    // After move finishes, check abort status and flags
    5:
        IF fbMotionStage.ExMotionStatus.bIdling THEN
            AssertTrue(
                Condition := fbMotionStage.ExMotionStatus.bAborted,
                Message   := 'Move must be aborted #8'
            );
            AssertFalse(
                Condition := fbMotionStage.stMotionStatus.bBusy,
                Message   := 'Move request must be canceled #9'
            );
            AssertFalse(
                Condition := fbMotionStage.stExMotionStatus.bExecute,
                Message   := 'Move request must cleared #10'
            );
            nTestStep := 6;
        END_IF	
END_CASE

// Cyclically call timer FBs
fbTestTimer();
fbAbsoluteMoveHaltTimer();

// End test or handle timeout
IF nTestStep = 6 THEN
    TEST_FINISHED();
ELSIF fbTestTimer.Q THEN
    AssertTrue(
        Condition := FALSE,
        Message := CONCAT('Timed out at step: ', TO_STRING(nTestStep))
    );
    TEST_FINISHED();
END_IF
END_METHOD

METHOD PRIVATE GivenMoveCmdAndMoveOkIfResetThenAbortMove_Test1
VAR_INST
   fbMotionStage : FB_MotionStageNC(	sName := 'TEST1',
                                        AxisRef := fbAxisRef[1],
                                        iPersistentDataStorage := fbPersistentDataStorage[1]
                                    ):=(SaveAxisParams := FALSE);
									
    fbTestTimer: TON := (IN:=TRUE, PT:=T#3S);
    fbAbsoluteMoveResetTimer: TON := (PT:=T#500MS);
    nTestStep : INT;
END_VAR
TEST(__POUNAME());

// motion stage block
fbMotionStage();

// Main test state machine
CASE nTestStep OF
    // === Interlock Fault Test ===
    0:
        IF fbMotionStage.ExMotionStatus.bInterlocksError THEN
            AssertTrue(
                Condition := fbMotionStage.stMotionStatus.bError,
                Message := 'Interlock error must be raised #1'
            );
            AssertEquals_UDINT(
                Expected := 11,
                Actual := fbMotionStage.stMotionStatus.nErrorId,
                Message := 'Interlock error code is 11 #2'
            );
        END_IF
        nTestStep := nTestStep + 1;
    
    // === Reset and Enable Features ===
    1:
        fbMotionStage.Reset();
        fbMotionStage.EnableLimits(
			BackwardEnable:=TRUE, 
			ForwardEnable:=TRUE,
			HomeEnable:=FALSE
		);
        fbMotionStage.EnableInterlocks();
        // Note: Trying to write to a property with 'GET' only should fail! See notes below.
        // fbMotionStage.MotionStatus.bExecute := TRUE; // Should be forbidden if it's a read-only property

        nTestStep := nTestStep + 1;    

    // === Abort Done/Status Check ===
    2:
        IF fbMotionStage.ExMotionStatus.bAbortDone THEN
            AssertFalse(
                Condition := fbMotionStage.stMotionStatus.bError,
                Message := 'Error must be cleared #3'
            );
            AssertEquals_UDINT(
                Expected := 0,
                Actual := fbMotionStage.stMotionStatus.nErrorId,
                Message := 'error ID must be 0 #4'
            );
            nTestStep := nTestStep + 1;    
        END_IF

    // === Absolute Move Request ===
    3:
        fbMotionStage.AbsoluteMove(
            Position := 10000.0,
            Velocity := 50.0,
            Acceleration := 500.0,
            Deceleration := 500.0
        );
        fbAbsoluteMoveResetTimer.IN := TRUE;
        nTestStep := nTestStep + 1;

    // === Move Reset after Timer ===
    4:
        IF fbAbsoluteMoveResetTimer.Q THEN
            fbMotionStage.Reset();
            fbAbsoluteMoveResetTimer.IN := FALSE;
            nTestStep := nTestStep + 1;
        END_IF

    // === Move Done/Abort Confirmation ===
    5:
        IF fbMotionStage.stExMotionStatus.bAbortDone THEN
            nTestStep := nTestStep + 1;
        END_IF
	6:
		IF fbMotionStage.stExMotionStatus.bAborted THEN
            AssertFalse(
                Condition := fbMotionStage.stMotionStatus.bBusy,
                Message := 'Move request must be canceled #6'
            );
            AssertFalse(
                Condition := fbMotionStage.stExMotionStatus.bExecute,
                Message := 'Move request must be cleared #7'
            );
            nTestStep := nTestStep + 1;
		END_IF
END_CASE

// Update timers
fbTestTimer();
fbAbsoluteMoveResetTimer();

// Test Completion Handlers
IF nTestStep = 7 THEN
    TEST_FINISHED();
ELSIF fbTestTimer.Q THEN
    AssertTrue(
        Condition := FALSE,
        Message := CONCAT('Timed out at step: ', TO_STRING(nTestStep))
    );
    TEST_FINISHED();
END_IF
END_METHOD

METHOD PRIVATE GivenMoveCmdAndMoveOkMoveToTarget1ThenTarget2_Test3
VAR_INST
   fbMotionStage : FB_MotionStageNC(	sName := 'Test3',
                                        AxisRef := fbAxisRef[3],
                                        iPersistentDataStorage := fbPersistentDataStorage[3]
                                    ):=(SaveAxisParams := FALSE);
									
    fbTestTimer: TON := (IN:=TRUE, PT:=T#10S);
    nTestStep : INT;
END_VAR
TEST(__POUNAME());

CASE nTestStep OF
    0: // Enable safety interlocks and hardware limits
        fbMotionStage.EnableLimits(
			BackwardEnable:=TRUE, 
			ForwardEnable:=TRUE,
			HomeEnable:=FALSE
		);
        fbMotionStage.EnableInterlocks();
        nTestStep := 1;

    1: // Issue initial absolute move to position 100.0 with no backlash
        fbMotionStage.AbsoluteMove(
            Position := 100.0,
            Velocity := 50.0,
            Acceleration := 500.0,
            Deceleration := 500.0
        );
        nTestStep := 2;

    2: // Wait for move done
        IF fbMotionStage.stMotionStatus.bDone THEN
            AssertTrue(
                Condition := ABS(fbMotionStage.MotionCmd.fPosition - fbAxisRef[3].NcToPlc.ActPos) < 0.001,
                Message := 'Target position not reached #1'
            );
            nTestStep := 3;
        END_IF

    3: // When idling, perform another absolute move
        IF fbMotionStage.ExMotionStatus.bIdling THEN
            fbMotionStage.AbsoluteMove(
                Position := 320.0,
                Velocity := 50.0,
                Acceleration := 500.0,
                Deceleration := 500.0
            );
            nTestStep := 4;
        END_IF

    4: // Wait for second move done
        IF fbMotionStage.stMotionStatus.bDone THEN
            AssertTrue(
                Condition := ABS(fbMotionStage.MotionCmd.fPosition - fbAxisRef[3].NcToPlc.ActPos) < 0.001,
                Message := 'Target position not reached #2'
            );
            nTestStep := 5;
          END_IF

END_CASE

fbTestTimer();
fbMotionStage();

IF nTestStep = 5 THEN
    TEST_FINISHED();
ELSIF fbTestTimer.Q THEN
    AssertTrue(
        Condition := FALSE,
        Message := CONCAT('Timed out at step: ', TO_STRING(nTestStep))
    );
    TEST_FINISHED();
END_IF
END_METHOD

METHOD PRIVATE GivenMoveCmdAndValidInterlocksThenMoveToTarget_Test4
VAR_INST
   fbMotionStage : FB_MotionStageNC(	sName := 'Test4',
                                        AxisRef := fbAxisRef[4],
                                        iPersistentDataStorage := fbPersistentDataStorage[4]
                                    ):=(SaveAxisParams := FALSE);
									
    fbTestTimer: TON := (IN:=TRUE, PT:=T#3S);
    nTestStep : INT;
END_VAR
TEST(__POUNAME());

CASE nTestStep OF
    0: // Enable safety interlocks and hardware limits
        fbMotionStage.EnableLimits(
			BackwardEnable:=TRUE, 
			ForwardEnable:=TRUE,
			HomeEnable:=FALSE
		);
        fbMotionStage.EnableInterlocks();
        nTestStep := 1;

    1: // Issue initial absolute move to position 100.0 with no backlash
        fbMotionStage.AbsoluteMove(
            Position := 100.0,
            Velocity := 50.0,
            Acceleration := 500.0,
            Deceleration := 500.0
        );
        nTestStep := 2;

    2: // Wait for move done
        IF fbMotionStage.stMotionStatus.bDone THEN
            AssertTrue(
                Condition := ABS(fbMotionStage.MotionCmd.fPosition - fbAxisRef[4].NcToPlc.ActPos) < 0.001,
                Message := 'Target position not reached #1'
            );
            nTestStep := 3;
        END_IF
END_CASE

fbTestTimer();
fbMotionStage();

IF nTestStep = 3 THEN
    TEST_FINISHED();
ELSIF fbTestTimer.Q THEN
    AssertTrue(
        Condition := FALSE,
        Message := CONCAT('Timed out at step: ', TO_STRING(nTestStep))
    );
    TEST_FINISHED();
END_IF
END_METHOD

METHOD PRIVATE GivenMoveCmdValidInterlockAndWrongMotionParamsThenGotoErrorStateIfResetThenGotoInitState_Test5
VAR_INST
   fbMotionStage : FB_MotionStageNC(	sName := 'Test5',
                                        AxisRef := fbAxisRef[5],
                                        iPersistentDataStorage := fbPersistentDataStorage[5]
                                    ):=(SaveAxisParams := FALSE);
									
    fbTestTimer: TON := (IN:=TRUE, PT:=T#3S);
    fbAbsoluteMoveTimer: TON := (PT:=T#50MS);
    nTestStep : INT;
END_VAR
TEST(__POUNAME());

CASE nTestStep OF
    0:
        fbMotionStage.EnableLimits(
			BackwardEnable:=TRUE, 
			ForwardEnable:=TRUE,
			HomeEnable:=FALSE
		);
        fbMotionStage.EnableInterlocks();
        nTestStep := 1;
	1:// Issue initial absolute move to position 100.0 with no backlash
        fbMotionStage.AbsoluteMove(
            Position := 100.0,
            Velocity := 0.0,
            Acceleration := 500.0,
            Deceleration := 500.0
        );
		nTestStep := 2;
	2:
		IF (fbMotionStage.stExMotionStatus.eDriveState=E_MoveState.ERROR) THEN
			nTestStep := 3;
		END_IF
END_CASE
fbMotionStage();
fbTestTimer();
fbAbsoluteMoveTimer();


IF nTestStep = 3 THEN

TEST_FINISHED();
ELSIF fbTestTimer.Q THEN
    AssertTrue(
        Condition := FALSE,
        Message := CONCAT('Timed out at step: ', TO_STRING(nTestStep))
    );
    TEST_FINISHED();
END_IF
END_METHOD

METHOD PRIVATE OverallStageFeaturesAndOperationalTests_Test17
VAR_INST
   fbMotionStage : FB_MotionStageNC(	sName := 'Test17',
                                        AxisRef := fbAxisRef[17],
                                        iPersistentDataStorage := fbPersistentDataStorage[17]
                                    ) := (SaveAxisParams := FALSE);
									
    fbTestTimer: TON := (IN:=TRUE, PT:=T#180S);
    fbResetTimer: TON := (IN:=FALSE, PT:=T#500MS);;
	fbInMotionTimer : TON := (IN:=FALSE, PT:=T#800MS);;
    fbCamSwitchPulserSearch : TON := (IN:=FALSE, PT:=T#1000MS);
    fbCamSwitchPulserSync: TON := (IN:=FALSE, PT:=T#2000MS);
    nTestStep : INT;
END_VAR
TEST(__POUNAME());

CASE nTestStep OF

/// ------------ INITIAL SETUP ---------------
0:
    fbMotionStage.EnableLimits(
        BackwardEnable := TRUE, ForwardEnable := TRUE, HomeEnable := FALSE);
    fbMotionStage.EnableInterlocks();
    nTestStep := 1;

/// ------- 3 FAST ABSOLUTE MOVES ------------
/// (All moves <= 50 units, velocities set for sub-second moves)
1:
    fbMotionStage.AbsoluteMove(Position := 10.0, Velocity := 50.0, Acceleration := 200.0, Deceleration := 200.0);
    nTestStep := 2;
2:
    IF fbMotionStage.stMotionStatus.bDone THEN
        AssertTrue(ABS(10.0 - fbAxisRef[17].NcToPlc.ActPos) < 0.01, 'Move#1');
        nTestStep := 3;
    END_IF
3:
    fbMotionStage.AbsoluteMove(Position := -8.0, Velocity := 50.0, Acceleration := 200.0, Deceleration := 200.0);
    nTestStep := 4;
4:
    IF fbMotionStage.stMotionStatus.bDone THEN
        AssertTrue(ABS(-8.0 - fbAxisRef[17].NcToPlc.ActPos) < 0.01, 'Move#2');
        nTestStep := 5;
    END_IF
5:
    fbMotionStage.AbsoluteMove(Position := 15.0, Velocity := 50.0, Acceleration := 150.0, Deceleration := 150.0);
    nTestStep := 6;
6:
    IF fbMotionStage.stMotionStatus.bDone THEN
        AssertTrue(ABS(15.0 - fbAxisRef[17].NcToPlc.ActPos) < 0.01, 'Move#3');
        nTestStep := 7;
    END_IF

/// -------- HALT and RESET POS/NEG ------------

7:
    fbMotionStage.AbsoluteMove(Position := 18.0, Velocity := 70.0, Acceleration := 200.0, Deceleration := 200.0);
    fbInMotionTimer.PT := T#120MS;
    fbInMotionTimer.IN := TRUE;
    nTestStep := 8;
8:
    IF fbMotionStage.stMotionStatus.bBusy AND fbInMotionTimer.Q THEN
        fbMotionStage.Halt();
        fbInMotionTimer.IN := FALSE;
        nTestStep := 9;
    END_IF
9:
    IF fbMotionStage.stExMotionStatus.bAborted THEN
        AssertFalse(fbMotionStage.stMotionStatus.bBusy, 'Halt busy/fwd');
        nTestStep := 10;
    END_IF

10:
    fbMotionStage.AbsoluteMove(Position := -12.0, Velocity := 70.0, Acceleration := 200.0, Deceleration := 200.0);
    fbInMotionTimer.PT := T#120MS;
    fbInMotionTimer.IN := TRUE;
    nTestStep := 11;
11:
    IF fbMotionStage.stMotionStatus.bBusy AND fbInMotionTimer.Q THEN
        fbMotionStage.Halt();
        fbInMotionTimer.IN := FALSE;
        nTestStep := 12;
    END_IF
12:
    IF fbMotionStage.stExMotionStatus.bAborted THEN
        AssertFalse(fbMotionStage.stMotionStatus.bBusy, 'Halt busy/bwd');
        nTestStep := 13;
    END_IF

13:
    fbMotionStage.AbsoluteMove(Position := 21.0, Velocity := 70.0, Acceleration := 200.0, Deceleration := 200.0);
    fbInMotionTimer.PT := T#120MS;
    fbInMotionTimer.IN := TRUE;
    nTestStep := 14;
14:
    IF fbMotionStage.stMotionStatus.bBusy AND fbInMotionTimer.Q THEN
        fbMotionStage.Reset();
        fbInMotionTimer.IN := FALSE;
        nTestStep := 15;
    END_IF
15:
    IF fbMotionStage.stExMotionStatus.bAborted THEN
        AssertFalse(fbMotionStage.stMotionStatus.bBusy, 'Reset busy/fwd');
        nTestStep := 16;
    END_IF

16:
    fbMotionStage.AbsoluteMove(Position := -22.0, Velocity := 70.0, Acceleration := 200.0, Deceleration := 200.0);
    fbInMotionTimer.PT := T#120MS;
    fbInMotionTimer.IN := TRUE;
    nTestStep := 17;
17:
    IF fbMotionStage.stMotionStatus.bBusy AND fbInMotionTimer.Q THEN
        fbMotionStage.Reset();
        fbInMotionTimer.IN := FALSE;
        nTestStep := 18;
    END_IF
18:
    IF fbMotionStage.stExMotionStatus.bAborted THEN
        AssertFalse(fbMotionStage.stMotionStatus.bBusy, 'Reset busy/bwd');
        nTestStep := 19;
    END_IF

/// -------- LIMIT HIT TEST (FORWARD THEN BACKWARD) ----------
19:
    fbMotionStage.AbsoluteMove(Position := 25.0, Velocity := 50.0, Acceleration := 120.0, Deceleration := 120.0);
    fbInMotionTimer.PT := T#120MS; fbInMotionTimer.IN := TRUE; nTestStep := 20;
20:
    IF fbMotionStage.stMotionStatus.bBusy AND fbInMotionTimer.Q THEN
        fbMotionStage.EnableLimits(BackwardEnable := TRUE, ForwardEnable := FALSE, HomeEnable := FALSE);
        fbInMotionTimer.IN := FALSE; nTestStep := 21;
    END_IF
21:
    IF fbMotionStage.stMotionStatus.bWarning AND fbMotionStage.stExMotionStatus.bAborted THEN
        fbMotionStage.EnableLimits(BackwardEnable := TRUE, ForwardEnable := TRUE, HomeEnable := FALSE);
        nTestStep := 22;
    END_IF
22: nTestStep := 23;

23:
    fbMotionStage.AbsoluteMove(Position := -25.0, Velocity := 50.0, Acceleration := 120.0, Deceleration := 120.0);
    fbInMotionTimer.PT := T#120MS; fbInMotionTimer.IN := TRUE; nTestStep := 24;
24:
    IF fbMotionStage.stMotionStatus.bBusy AND fbInMotionTimer.Q THEN
        fbMotionStage.EnableLimits(BackwardEnable := FALSE, ForwardEnable := TRUE, HomeEnable := FALSE);
        fbInMotionTimer.IN := FALSE; nTestStep := 25;
    END_IF
25:
    IF fbMotionStage.stMotionStatus.bWarning AND fbMotionStage.stExMotionStatus.bAborted THEN
        fbMotionStage.EnableLimits(BackwardEnable := TRUE, ForwardEnable := TRUE, HomeEnable := FALSE);
        nTestStep := 26;
    END_IF
26: nTestStep := 27;

/// ------------- Home+Move Alternation: All major home modes ------------
/// (Home, then absolute move. All positions ~10-30 units, velocities >= 50.)
27:
    fbMotionStage.Home(HomePosition := 10.0, HomeMode := E_EpicsHomeCmd.LOW_LIMIT);
    fbCamSwitchPulserSearch.IN := TRUE; nTestStep := 28;
28:
    IF fbCamSwitchPulserSearch.Q THEN
        fbMotionStage.EnableLimits(BackwardEnable := FALSE, ForwardEnable := TRUE, HomeEnable := FALSE);
        fbCamSwitchPulserSearch.IN := FALSE; fbCamSwitchPulserSync.IN := TRUE;
        nTestStep := 29;
    END_IF
29:
    IF fbCamSwitchPulserSync.Q THEN
        fbMotionStage.EnableLimits(BackwardEnable := TRUE, ForwardEnable := TRUE, HomeEnable := FALSE);
        fbCamSwitchPulserSync.IN := FALSE; nTestStep := 30;
    END_IF
30:
    IF fbMotionStage.stMotionStatus.bDone THEN
        AssertTrue(fbAxisRef[17].Status.Homed, 'Home#1 (LOW_LIMIT): Axis not calibrated'); 
		AssertEquals_LREAL(Delta := 0.001, Expected := 10.0, Actual := fbAxisRef[17].NcToPlc.ActPos, Message :='Home#1: Not at expected home');
        nTestStep := 31;
    END_IF
31: 
	fbMotionStage.AbsoluteMove(Position := 20.0, Velocity := 50.0, Acceleration := 200.0, Deceleration := 200.0);
	nTestStep := 32;
32: 
	IF fbMotionStage.stMotionStatus.bDone THEN
		AssertTrue(ABS(20.0 - fbAxisRef[17].NcToPlc.ActPos) < 0.01, 'Move#4: Target position not reached after home');
		nTestStep := 33;
	END_IF

33: 
	fbMotionStage.Home(HomePosition := 25.0, HomeMode := E_EpicsHomeCmd.HIGH_LIMIT);
	fbCamSwitchPulserSearch.IN := TRUE; 
	nTestStep := 34;
34: 
	IF fbCamSwitchPulserSearch.Q THEN 
		fbMotionStage.EnableLimits(BackwardEnable := TRUE, ForwardEnable := FALSE, HomeEnable := FALSE);
		fbCamSwitchPulserSearch.IN := FALSE;
		fbCamSwitchPulserSync.IN := TRUE;
		nTestStep := 35;
	END_IF
35: 
	IF fbCamSwitchPulserSync.Q THEN
		fbMotionStage.EnableLimits(BackwardEnable := TRUE, ForwardEnable := TRUE, HomeEnable := FALSE);
		fbCamSwitchPulserSync.IN := FALSE;
		nTestStep := 36;
	END_IF
36: 
	IF fbMotionStage.stMotionStatus.bDone THEN 
		AssertTrue(fbAxisRef[17].Status.Homed, 'Home#2 (HIGH_LIMIT): Axis not calibrated');
		AssertEquals_LREAL(Delta := 0.001, Expected := 25.0, Actual := fbAxisRef[17].NcToPlc.ActPos, Message := 'Home#2: Not at expected home'); 
		nTestStep := 37; 
	END_IF
37: 
	fbMotionStage.AbsoluteMove(Position := -20.0, Velocity := 50.0, Acceleration := 200.0, Deceleration := 200.0); 
	nTestStep := 38;
38: 
	IF fbMotionStage.stMotionStatus.bDone THEN 
		AssertTrue(ABS(-20.0 - fbAxisRef[17].NcToPlc.ActPos) < 0.01, 'Move#5: Target position not reached after home');
		nTestStep := 39; 
	END_IF

39:
    fbMotionStage.Home(HomePosition := 12.0, HomeMode := E_EpicsHomeCmd.HOME_VIA_LOW);
    fbCamSwitchPulserSearch.IN := TRUE; nTestStep := 40;
40: 
	IF fbCamSwitchPulserSearch.Q THEN 
		fbMotionStage.EnableLimits(BackwardEnable := FALSE, ForwardEnable := TRUE, HomeEnable := FALSE); 
		fbCamSwitchPulserSearch.IN := FALSE; 
		fbCamSwitchPulserSync.IN := TRUE; 
		nTestStep := 41; 
	END_IF
41: 
	IF fbCamSwitchPulserSync.Q THEN
		fbMotionStage.EnableLimits(BackwardEnable := TRUE, ForwardEnable := TRUE, HomeEnable := FALSE);
		fbCamSwitchPulserSync.IN := FALSE;
		fbCamSwitchPulserSearch.IN := TRUE;
		nTestStep := 42;
	END_IF
42: 
	IF fbCamSwitchPulserSearch.Q THEN
		fbMotionStage.EnableLimits(BackwardEnable := TRUE, ForwardEnable := TRUE, HomeEnable := TRUE);
		fbCamSwitchPulserSearch.IN := FALSE;
		fbCamSwitchPulserSync.IN := TRUE;
		nTestStep := 43;
	END_IF
43: 
	IF fbCamSwitchPulserSync.Q THEN 
		fbMotionStage.EnableLimits(BackwardEnable := TRUE, ForwardEnable := TRUE, HomeEnable := FALSE);
		fbCamSwitchPulserSync.IN := FALSE; 
		nTestStep := 44; 
	END_IF
44: 
	IF fbMotionStage.stMotionStatus.bDone THEN 
		AssertTrue(fbAxisRef[17].Status.Homed, 'Home#3 (HOME_VIA_LOW): Axis not calibrated'); 
		AssertEquals_LREAL(Delta := 0.001, Expected := 12.0, Actual := fbAxisRef[17].NcToPlc.ActPos, Message := 'Home#3: Not at expected home');
		nTestStep := 45; 
	END_IF
45: 
	fbMotionStage.AbsoluteMove(Position := 25.0, Velocity := 50.0, Acceleration := 200.0, Deceleration := 200.0); 
	nTestStep := 46;
46: 
	IF fbMotionStage.stMotionStatus.bDone THEN 
		AssertTrue(ABS(25.0 - fbAxisRef[17].NcToPlc.ActPos) < 0.01, 'Move#6: Target position not reached after home');
		nTestStep := 47; 
	END_IF

47:
    fbMotionStage.Home(HomePosition := -15.0, HomeMode := E_EpicsHomeCmd.HOME_VIA_HIGH);
    fbCamSwitchPulserSearch.IN := TRUE; nTestStep := 48;
48: 
	IF fbCamSwitchPulserSearch.Q THEN 
		fbMotionStage.EnableLimits(BackwardEnable := TRUE, ForwardEnable := FALSE, HomeEnable := FALSE);
		fbCamSwitchPulserSearch.IN := FALSE;
		fbCamSwitchPulserSync.IN := TRUE;
		nTestStep := 49; 
	END_IF
49: 
	IF fbCamSwitchPulserSync.Q THEN 
		fbMotionStage.EnableLimits(BackwardEnable := TRUE, ForwardEnable := TRUE, HomeEnable := FALSE);
		fbCamSwitchPulserSync.IN := FALSE;
		fbCamSwitchPulserSearch.IN := TRUE;
		nTestStep := 50;
	END_IF
50: 
	IF fbCamSwitchPulserSearch.Q THEN
		fbMotionStage.EnableLimits(BackwardEnable := TRUE, ForwardEnable := TRUE, HomeEnable := TRUE);
		fbCamSwitchPulserSearch.IN := FALSE;
		fbCamSwitchPulserSync.IN := TRUE;
		nTestStep := 51;
	END_IF
51: 
	IF fbCamSwitchPulserSync.Q THEN 
		fbMotionStage.EnableLimits(BackwardEnable := TRUE, ForwardEnable := TRUE, HomeEnable := FALSE);
		fbCamSwitchPulserSync.IN := FALSE;
		nTestStep := 52; 
	END_IF
52: 
	IF fbMotionStage.stMotionStatus.bDone THEN 
		AssertTrue(fbAxisRef[17].Status.Homed, 'Home#4 (HOME_VIA_HIGH): Axis not calibrated');
		AssertEquals_LREAL(Delta := 0.001, Expected := -15.0, Actual := fbAxisRef[17].NcToPlc.ActPos, Message := 'Home#4: Not at expected home');
		nTestStep := 53; 
	END_IF
53: 
	fbMotionStage.AbsoluteMove(Position := -30.0, Velocity := 50.0, Acceleration := 200.0, Deceleration := 200.0);
	nTestStep := 54;
54: 
	IF fbMotionStage.stMotionStatus.bDone THEN 
		AssertTrue(ABS(-30.0 - fbAxisRef[17].NcToPlc.ActPos) < 0.01, 'Move#7: Target position not reached after home'); 
		nTestStep := 55;
	END_IF

55:
    fbMotionStage.Home(HomePosition := 30.0, HomeMode := E_EpicsHomeCmd.ABSOLUTE_SET); 
    nTestStep := 56;
56: 
	IF fbMotionStage.stMotionStatus.bDone THEN 
		AssertTrue(fbAxisRef[17].Status.Homed, 'Home#5 (ABSOLUTE_SET): Axis not calibrated'); 
		AssertEquals_LREAL(Delta := 0.001, Expected := 30.0, Actual := fbAxisRef[17].NcToPlc.ActPos,  Message := 'Home#5: Not at expected home');
		nTestStep := 57; 
	END_IF
57: 
	fbMotionStage.AbsoluteMove(Position := 23.0, Velocity := 50.0, Acceleration := 200.0, Deceleration := 200.0);
	nTestStep := 58;
58: 
	IF fbMotionStage.stMotionStatus.bDone THEN 
		AssertTrue(ABS(23.0 - fbAxisRef[17].NcToPlc.ActPos) < 0.01, 'Move#8: Target position not reached after home');
		nTestStep := 59;
	END_IF

// ---- Backlash Compensation: absolute moves ----
59: 
	fbMotionStage.EnableBacklashCompensation(UserEnable := TRUE, Compensation := 1.2);
	nTestStep := 60;
60: 
	fbMotionStage.AbsoluteMove(Position := 27.5, Velocity := 50.0, Acceleration := 100.0, Deceleration := 100.0);
	nTestStep := 61;
61: 
	IF fbMotionStage.stMotionStatus.bDone THEN 
        AssertTrue(ABS(27.5 - fbAxisRef[17].NcToPlc.ActPos) < 0.01, 'Move#9:No comp fwd expected');
        AssertTrue((fbAxisRef[17].NcToPlc.ActPos - fbAxisRef[17].NcToPlc.ActPosWithoutPosCorrection) = 0.0, 'No compensation in this direction');
        nTestStep := 62; 
    END_IF
62: 
	fbMotionStage.AbsoluteMove(Position := 21.0, Velocity := 50.0, Acceleration := 100.0, Deceleration := 100.0);
	nTestStep := 63;
63: 
	IF fbMotionStage.stMotionStatus.bDone THEN 
        AssertTrue(ABS(21.0 - fbAxisRef[17].NcToPlc.ActPos) < 0.01, 'Move#10: Target not reached'); 
        AssertTrue(((fbAxisRef[17].NcToPlc.ActPos - fbAxisRef[17].NcToPlc.ActPosWithoutPosCorrection)-1.2) < 0.001, 
                   'Compensation 1.2 not applied in reverse'); 
        nTestStep := 64; 
    END_IF
64: 
	fbMotionStage.EnableBacklashCompensation(UserEnable := FALSE, Compensation := 0.0);
	nTestStep := 65;
65: 
	fbMotionStage.AbsoluteMove(Position := -20.0, Velocity := 50.0, Acceleration := 100.0, Deceleration := 100.0);
	nTestStep := 66;
66: 
	IF fbMotionStage.stMotionStatus.bDone THEN 
        AssertTrue(ABS(-20.0 - fbAxisRef[17].NcToPlc.ActPos) < 0.01, 'Move#11: Target not reached (no comp)'); 
        AssertTrue((fbAxisRef[17].NcToPlc.ActPos - fbAxisRef[17].NcToPlc.ActPosWithoutPosCorrection) = 0.0, 'Compensation should be disabled'); 
        nTestStep := 67; 
    END_IF
67: 
	fbMotionStage.EnableBacklashCompensation(UserEnable := TRUE, Compensation := -1.7);
	nTestStep := 68;
68: 
	fbMotionStage.AbsoluteMove(Position := -30.0, Velocity := 50.0, Acceleration := 100.0, Deceleration := 100.0);
	nTestStep := 69;
69: 
	IF fbMotionStage.stMotionStatus.bDone THEN 
        AssertTrue(ABS(-30.0 - fbAxisRef[17].NcToPlc.ActPos) < 0.01, 'Move#12: Target not reached, comp negative'); 
        AssertTrue((fbAxisRef[17].NcToPlc.ActPos - fbAxisRef[17].NcToPlc.ActPosWithoutPosCorrection) = 0.0, 'No comp fwd for neg setting'); 
        nTestStep := 70; 
    END_IF
70: 
	fbMotionStage.AbsoluteMove(Position := 5.0, Velocity := 50.0, Acceleration := 100.0, Deceleration := 100.0);
	nTestStep := 71;
71: 
	IF fbMotionStage.stMotionStatus.bDone THEN 
        AssertTrue(ABS(5.0 - fbAxisRef[17].NcToPlc.ActPos) < 0.01, 'Move#13: Target not reached (comp negative, rev)'); 
        AssertTrue(((fbAxisRef[17].NcToPlc.ActPos - fbAxisRef[17].NcToPlc.ActPosWithoutPosCorrection)-1.7) < 0.001, 'Compensation -1.7 not applied'); 
        nTestStep := 72; 
    END_IF
72:
	fbMotionStage.EnableBacklashCompensation(UserEnable := FALSE, Compensation := 0.0);
	nTestStep := 73;
// --- Absolute Move with ZERO Velocity triggers error ---
73:
    fbMotionStage.AbsoluteMove(
        Position := 10.0,
        Velocity := 0.0,
        Acceleration := 100.0,
        Deceleration := 100.0
    );
    nTestStep := 74;

74:
    IF fbMotionStage.stMotionStatus.bError THEN
        AssertTrue(
            fbMotionStage.stMotionStatus.nErrorId = 16#4359,
            'Not the expected NC error message for zero velocity'
        );
        fbMotionStage.Reset();
        nTestStep := 75;
    END_IF

75:
    IF NOT fbMotionStage.stMotionStatus.bError THEN
        AssertFalse(
            fbMotionStage.stMotionStatus.bError,
            'Error flag should be cleared after reset'
        );
        AssertTrue(
            fbMotionStage.stMotionStatus.sErrorMessage = '',
            'Error message should be cleared after reset'
        );
        nTestStep := 76;
    END_IF

76:
    fbMotionStage.AbsoluteMove(
        Position := 15.0,
        Velocity := 50.0,
        Acceleration := 100.0,
        Deceleration := 100.0
    );
    nTestStep := 77;

77:
    IF fbMotionStage.stMotionStatus.bDone THEN
        AssertTrue(
            ABS(15.0 - fbAxisRef[17].NcToPlc.ActPos) < 0.01,
            'Recovery Move: Target position not reached after valid velocity'
        );
        nTestStep := 78;
    END_IF
END_CASE

fbCamSwitchPulserSearch();
fbCamSwitchPulserSync();
fbInMotionTimer();
fbTestTimer();
fbMotionStage();

IF nTestStep = 78 THEN
    TEST_FINISHED();
ELSIF fbTestTimer.Q THEN
    AssertTrue(FALSE, CONCAT('Timed out at step: ', TO_STRING(nTestStep)));
    TEST_FINISHED();
END_IF
END_METHOD

END_FUNCTION_BLOCK

// ---- Test/Interlok/FB_MotionInterlocksCommon_Test.TcPOU
FUNCTION_BLOCK FB_MotionInterlocksCommon_Test EXTENDS FB_TestSuite
VAR
    fbMotionLogger 		: ARRAY[1..5] OF FB_MotionLogger_TestDouble;
END_VAR

GivenEpicsEnableAndHardwareEnableIfNotUserEnableThenResetPowerEnableAndMoveOk_Test1();
GivenEpicsEnablehardwareEnableAndUserEnableUpdatePowerEnableAndMoveOk_Test2();
GivenhardwareEnableAndUserEnableIfNotEpicsEnableResetPowerEnable_Test3();
GivenUserEnableAndNothardwareEnableThenSetHardwareEnableErrorResetMoveOk_Test4();
GivenInterlockEventIFGlobalResetClearErrors_Test5();

METHOD PRIVATE GivenEpicsEnableAndHardwareEnableIfNotUserEnableThenResetPowerEnableAndMoveOk_Test1
VAR
    fbMotionInterlocksCommon : FB_MotionInterlocksCommon(
		iMotionLogger:=fbMotionLogger[1]
	);
    sExpectedUserEnableMessage : STRING := 'User enable interlock triggered!';
    sActUserEnableMessage : STRING;
END_VAR
TEST(__POUNAME());
// Test UserEnable interlock trigger
fbMotionInterlocksCommon.EnableInterlocks(UserEnable:=FALSE, HardwareEnable:=TRUE);
fbMotionInterlocksCommon.DriveCommands(MoveEnable:=TRUE, NewMoveReq:=FALSE);
fbMotionInterlocksCommon();

AssertFalse(Condition := fbMotionInterlocksCommon.PowerEnabled,
           Message := 'UserEnbale Interlock triggered PowerEnable must be unset #1');

AssertFalse(Condition := fbMotionInterlocksCommon.MoveOk,
           Message := 'UserEnbale Interlock triggered MoveOk must be unset #2');

sActUserEnableMessage := fbMotionInterlocksCommon.Message;
AssertEquals ( Expected:=sExpectedUserEnableMessage, Actual:=sActUserEnableMessage,
            Message:='Incorrect UserEnbale trigger Error Msg #3');

TEST_FINISHED();
END_METHOD

METHOD PRIVATE GivenEpicsEnablehardwareEnableAndUserEnableUpdatePowerEnableAndMoveOk_Test2
VAR
    fbMotionInterlocksCommon : FB_MotionInterlocksCommon(
		iMotionLogger:=fbMotionLogger[2]
	);
    sExpectedMessage : STRING := '';
    sActMessage : STRING;
    nExpectedErrorId : UDINT := 0;
    nActErrorId : UDINT;
END_VAR
TEST(__POUNAME());
// PowerEnable and MoveOk Set
fbMotionInterlocksCommon.EnableInterlocks(UserEnable:=TRUE, HardwareEnable:=TRUE);
fbMotionInterlocksCommon.DriveCommands(MoveEnable:=TRUE, NewMoveReq:=FALSE);
fbMotionInterlocksCommon();

AssertTrue(Condition := fbMotionInterlocksCommon.PowerEnabled,
           Message := 'Hardware or UserEnable Interlock not set #1');

AssertTrue(Condition := fbMotionInterlocksCommon.MoveOk,
           Message := 'Hardware or UserEnable Interlock not set #2');

AssertFalse(Condition := fbMotionInterlocksCommon.Error,
           Message := 'No Error expected #3');

nActErrorId := fbMotionInterlocksCommon.ErrorID;
AssertEquals ( Expected:=nExpectedErrorId, Actual:=nActErrorId ,
            Message:='ErrorID must be 0 #4');

sActMessage := fbMotionInterlocksCommon.Message;
AssertEquals ( Expected:=sExpectedMessage, Actual:=sActMessage ,
            Message:='No error Message #5');

TEST_FINISHED();
END_METHOD

METHOD PRIVATE GivenhardwareEnableAndUserEnableIfNotEpicsEnableResetPowerEnable_Test3
VAR
    fbMotionInterlocksCommon : FB_MotionInterlocksCommon(
		iMotionLogger:=fbMotionLogger[3]
	);
    sExpectedMessage : STRING := '';
    sActMessage : STRING;
    nExpectedErrorId : UDINT := 0;
    nActErrorId : UDINT;
END_VAR
TEST(__POUNAME());

fbMotionInterlocksCommon.EnableInterlocks(UserEnable:=TRUE, HardwareEnable:=TRUE);
fbMotionInterlocksCommon.DriveCommands(MoveEnable:=FALSE, NewMoveReq:=FALSE);
fbMotionInterlocksCommon();

AssertFalse(Condition := fbMotionInterlocksCommon.PowerEnabled,
           Message := 'No Epics Enable, PowerEnabled must not be set #1');

AssertTrue(Condition := fbMotionInterlocksCommon.MoveOk,
           Message := 'Epics Enable reset, Move Request must be invalid #2');

AssertFalse(Condition := fbMotionInterlocksCommon.Error,
           Message := 'No Error expected #3');

nActErrorId := fbMotionInterlocksCommon.ErrorID;
AssertEquals ( Expected:=nExpectedErrorId, Actual:=nActErrorId ,
            Message:='ErrorID must be 0 #4');

sActMessage := fbMotionInterlocksCommon.Message;
AssertEquals ( Expected:=sExpectedMessage, Actual:=sActMessage ,
            Message:='No error Message #5');
TEST_FINISHED();
END_METHOD

METHOD PRIVATE GivenInterlockEventIFGlobalResetClearErrors_Test5
VAR
     fbMotionInterlocksCommon : FB_MotionInterlocksCommon(
		iMotionLogger:=fbMotionLogger[5]
	);
    sExpectedMessage : STRING := '';
    sActMessage : STRING;
    nExpectedErrorId : UDINT := 0;
    nActErrorId : UDINT;
END_VAR
TEST(__POUNAME());
// HardwareEnable unset
fbMotionInterlocksCommon.EnableInterlocks(UserEnable:=TRUE, HardwareEnable:=FALSE);
fbMotionInterlocksCommon.DriveCommands(MoveEnable:=FALSE, NewMoveReq:=FALSE);
fbMotionInterlocksCommon();

AssertTRUE(Condition := fbMotionInterlocksCommon.Error,
           Message := 'HardwareEnable Error must be set #1');

// Test Global Reset to clear internal flags
fbMotionInterlocksCommon.EnableInterlocks(UserEnable:=TRUE, HardwareEnable:=TRUE);
fbMotionInterlocksCommon.Reset();
fbMotionInterlocksCommon();

AssertFalse(Condition := fbMotionInterlocksCommon.Error,
           Message := 'Error must be clear after global reset #2');

sActMessage := fbMotionInterlocksCommon.Message;
AssertEquals ( Expected:=sExpectedMessage, Actual:=sActMessage,
            Message:='Error Msg must be cleared #3');
TEST_FINISHED();
END_METHOD

METHOD PRIVATE GivenUserEnableAndNothardwareEnableThenSetHardwareEnableErrorResetMoveOk_Test4
VAR
    fbMotionInterlocksCommon : FB_MotionInterlocksCommon(
		iMotionLogger:=fbMotionLogger[4]
	);
    sExpectedHardwareEnableMessage : STRING := 'Hardware enable interlock triggered!';
    sActHardwareEnableMessage : STRING;
    nExpectedErrorId : UDINT := 11;
    nActErrorId : UDINT;
END_VAR
TEST(__POUNAME());
// HardwareEnable unset
fbMotionInterlocksCommon.EnableInterlocks(UserEnable:=TRUE, HardwareEnable:=FALSE);
fbMotionInterlocksCommon.DriveCommands(MoveEnable:=TRUE, NewMoveReq:=FALSE);
fbMotionInterlocksCommon();
// 
AssertFalse(Condition := fbMotionInterlocksCommon.PowerEnabled,
           Message := 'Hardware Interlock triggered PowerEnable must be unset #1');

AssertFalse(Condition := fbMotionInterlocksCommon.MoveOk,
           Message := 'Hardware Interlock triggered MoveOk must be unset #2');
// 
AssertTrue(Condition := fbMotionInterlocksCommon.Error,
           Message := 'Hardware Interlock triggered Error must be set #3');

AssertTrue(condition:=nExpectedErrorId = fbMotionInterlocksCommon.ErrorID, Message:='Incorrect Hardware trigger ErrorID #4');

AssertTrue ( condition:=(fbMotionInterlocksCommon.Message = sExpectedHardwareEnableMessage) , Message:='Incorrect Hardware trigger Error Msg #5');

TEST_FINISHED();
END_METHOD

END_FUNCTION_BLOCK

// ---- Test/TestDouble/FB_MotionLogger_TestDouble.TcPOU
FUNCTION_BLOCK FB_MotionLogger_TestDouble IMPLEMENTS I_MotionLogger
VAR
END_VAR

{warning 'Add method implementation '}
METHOD Clear
END_METHOD

METHOD ErrorCodeLookup : STRING
VAR_INPUT
	nErrorId	: UDINT;
END_VAR
END_METHOD

METHOD GetAllMessages :  STRING(1024)
END_METHOD

{warning 'Add method implementation '}
METHOD GetMessageCount : UINT
VAR_OUTPUT
	nCount	: UINT;
END_VAR
END_METHOD

{warning 'Add method implementation '}
METHOD Logger
VAR_INPUT
	Message	: STRING;
	Level	: E_MotionLogLevel := .E_MotionLogLevel.INFO;
	Source	: STRING := '';
END_VAR
END_METHOD

{warning 'Add property implementation'}
PROPERTY Name : STRING
GET
END_GET
END_PROPERTY

END_FUNCTION_BLOCK

// ---- Test/Interlok/FB_MotionInterlocksLimSw_Test.TcPOU
FUNCTION_BLOCK INTERNAL FB_MotionInterlocksLimSw_Test EXTENDS FB_TestSuite
VAR
    fbLimSwStatus: ARRAY [1..6] OF FB_LimSwStatus_testDouble;
    fbMotionInterlocksCommon:  ARRAY [1..6] OF  FB_MotionInterlocksCommon_TestDouble;
    fbMotionLogger : ARRAY [1..16] OF FB_MotionLogger_TestDouble;
END_VAR

GivenPositiveLimHitEventIfGlobalResetOrNewMoveReqClearLocalFlags_Test1();
GivenLimSwStatusEventIfStandStillUpdateBackwardAndFowardEnable_Test2();
GivenCommonInterlockErrorsThenSetLocalErrors_Test3();
GivenLimForwardAndBackwardActiveAxisMovingInNegativeDirectionIfPosiveLimishitThenNoLimHitEvent_Test4();
GivenLimForwardAndBackwardActiveAxisMovingInPosiveDirectionIfPosiveLimishitThenLimHitEventOccured_test5();
GivenLimSwStatusActiveAndAxisHomingInPosOrNegDirectionThenNoLimHitEvent_Test6();

METHOD PRIVATE GivenCommonInterlockErrorsThenSetLocalErrors_Test3
VAR_INST
    nExpectedErrorId: UDINT := 1;
    nActErrorId: UDINT;
    sExpectedMessage: STRING := 'User enable interlock triggered!';
    sActMessage: STRING;
    // subject under test
    fbMotionInterlocksLimSw : FB_MotionInterlocksLimSw(
		iMotionInterlocksCommon:=fbMotionInterlocksCommon[3], 
		iLimSwStatus:=fbLimSwStatus[3],
		iMotionLogger := fbMotionLogger[3]
	);
END_VAR
TEST(__POUNAME());
// Test UserEnable interlock trigger
fbMotionInterlocksCommon[3].Error := TRUE;
fbMotionInterlocksCommon[3].ErrorID:=1;
fbMotionInterlocksCommon[3].Message:=sExpectedMessage;
fbMotionInterlocksCommon[3]();
fbMotionInterlocksLimSw();

AssertTrue(Condition := fbMotionInterlocksLimSw.Error,
           Message := 'Common interlock event must set this error #1');

nActErrorId := fbMotionInterlocksLimSw.ErrorID;
AssertEquals ( Expected:=nExpectedErrorId, Actual:=nActErrorId ,
            Message:='Common interlock event must set this errorId #2');

sActMessage := fbMotionInterlocksLimSw.Message;
AssertEquals ( Expected:=sExpectedMessage, Actual:=sActMessage,
            Message:='Common interlock event must set this error msg #3');

fbMotionInterlocksCommon[3].ResetErrors();
fbMotionInterlocksCommon[3]();
fbMotionInterlocksLimSw();

TEST_FINISHED();
END_METHOD

METHOD PRIVATE GivenLimForwardAndBackwardActiveAxisMovingInNegativeDirectionIfPosiveLimishitThenNoLimHitEvent_Test4
VAR_INST
    tonLimSwStatusEvent : TON := (IN:=TRUE, PT:=T#0S);
    fbMotionInterlocksLimSw : FB_MotionInterlocksLimSw(
		iMotionInterlocksCommon:=fbMotionInterlocksCommon[4], 
		iLimSwStatus:=fbLimSwStatus[4],
		iMotionLogger := fbMotionLogger[4]
	);
END_VAR
TEST(__POUNAME());
tonLimSwStatusEvent();
fbLimSwStatus[4].LimitForwardEnable := TRUE;
fbLimSwStatus[4].LimitBackwardEnable := TRUE;
fbLimSwStatus[4]();
fbMotionInterlocksLimSw.AxisStatus(HomeBusy:=FALSE, PositiveDirection:=FALSE, NegativeDirection:=TRUE);
fbMotionInterlocksLimSw();


IF tonLimSwStatusEvent.Q THEN
    fbLimSwStatus[4].LimitForwardEnable := FALSE;
    fbLimSwStatus[4]();
    tonLimSwStatusEvent.IN:=FALSE;
END_IF

fbMotionInterlocksLimSw();

AssertFalse(Condition := fbMotionInterlocksLimSw.Warning,
           Message := 'No Warning event expected #1');
AssertFalse(Condition := fbMotionInterlocksLimSw.Warning,
           Message := 'No Lim Hit event expected #2');
TEST_FINISHED();
END_METHOD

METHOD PRIVATE  GivenLimForwardAndBackwardActiveAxisMovingInPosiveDirectionIfPosiveLimishitThenLimHitEventOccured_Test5
VAR_INST
    tonLimSwStatusEvent : TON := (IN:=TRUE, PT:=T#0S);
    fbMotionInterlocksLimSw : FB_MotionInterlocksLimSw(
		iMotionInterlocksCommon:=fbMotionInterlocksCommon[5], 
		iLimSwStatus:=fbLimSwStatus[5],
		iMotionLogger := fbMotionLogger[5]
	);
END_VAR
TEST(__POUNAME());
tonLimSwStatusEvent();
fbLimSwStatus[5].LimitForwardEnable := TRUE;
fbLimSwStatus[5].LimitBackwardEnable := TRUE;
fbMotionInterlocksLimSw.AxisStatus(HomeBusy:=FALSE, PositiveDirection:=TRUE, NegativeDirection:=FALSE);
fbLimSwStatus[5]();
fbMotionInterlocksLimSw();

IF tonLimSwStatusEvent.Q THEN
    fbLimSwStatus[5].LimitForwardEnable := FALSE;
    tonLimSwStatusEvent.IN := FALSE;
END_IF

fbLimSwStatus[5]();
fbMotionInterlocksLimSw();

AssertTrue(Condition := fbMotionInterlocksLimSw.Warning,
                   Message := 'Expecting a Warning event after positive lim hit #1');
AssertTrue(Condition := fbMotionInterlocksLimSw.Warning,
                   Message := 'Expecting a Limit hit event after positive lim hit #2');
TEST_FINISHED();
END_METHOD

METHOD PRIVATE GivenLimSwStatusActiveAndAxisHomingInPosOrNegDirectionThenNoLimHitEvent_Test6
VAR_INST
    fbMotionInterlocksLimSw : FB_MotionInterlocksLimSw(
		iMotionInterlocksCommon:=fbMotionInterlocksCommon[6], 
		iLimSwStatus:=fbLimSwStatus[6],
		iMotionLogger := fbMotionLogger[6]
	);
END_VAR
TEST(__POUNAME());

fbLimSwStatus[6].LimitForwardEnable := TRUE;
fbLimSwStatus[6].LimitBackwardEnable := TRUE;
fbMotionInterlocksLimSw.AxisStatus(HomeBusy:=TRUE, PositiveDirection:=TRUE, NegativeDirection:=FALSE);
fbLimSwStatus[6]();
fbMotionInterlocksLimSw();

AssertFalse(Condition := fbMotionInterlocksLimSw.Warning,
           Message := 'Warning event while homing unexpected #1');

AssertFalse(Condition := fbMotionInterlocksLimSw.Warning,
           Message := 'Lim hit event while homing unexpected #2');

fbMotionInterlocksLimSw.AxisStatus(HomeBusy:=TRUE, PositiveDirection:=FALSE, NegativeDirection:=TRUE);
fbLimSwStatus[6]();
fbMotionInterlocksLimSw();

AssertFalse(Condition := fbMotionInterlocksLimSw.Warning,
           Message := 'Warning event while homing unexpected #3');

AssertFalse(Condition := fbMotionInterlocksLimSw.Warning,
           Message := 'Lim hit event while homing unexpected #4');

TEST_FINISHED();
END_METHOD

METHOD PRIVATE GivenLimSwStatusEventIfStandStillUpdateBackwardAndFowardEnable_Test2
VAR_INST
    fbMotionInterlocksLimSw : FB_MotionInterlocksLimSw(
		iMotionInterlocksCommon:=fbMotionInterlocksCommon[2], 
		iLimSwStatus:=fbLimSwStatus[2],
		iMotionLogger := fbMotionLogger[2]
	);
END_VAR
TEST(__POUNAME());
// Test LimSwStatus Events and update backward and forward Enable
fbLimSwStatus[2].LimitForwardEnable := TRUE;
fbLimSwStatus[2].LimitBackwardEnable := TRUE;
fbMotionInterlocksLimSw.AxisStatus(HomeBusy:=FALSE, PositiveDirection:=FALSE, NegativeDirection:=FALSE);
fbLimSwStatus[2]();
fbMotionInterlocksLimSw();

AssertTrue(Condition := fbMotionInterlocksLimSw.MoveBackwardEnabled,
           Message := 'MoveBackwardEnabled must be set #1');

AssertTrue(Condition := fbMotionInterlocksLimSw.MoveForwardEnabled,
           Message := 'MoveForwardwardEnabled must be set #2');

fbLimSwStatus[2].LimitForwardEnable := FALSE;
fbLimSwStatus[2].LimitBackwardEnable := FALSE;
fbMotionInterlocksLimSw.AxisStatus(HomeBusy:=FALSE, PositiveDirection:=FALSE, NegativeDirection:=FALSE);
fbLimSwStatus[2]();
fbMotionInterlocksLimSw();

AssertFalse(Condition := fbMotionInterlocksLimSw.MoveBackwardEnabled,
           Message := 'MoveBackwardEnabled must not be set #3');

AssertFalse(Condition := fbMotionInterlocksLimSw.MoveForwardEnabled,
           Message := 'MoveForwardwardEnabled must not be set #4');

TEST_FINISHED();
END_METHOD

METHOD PRIVATE GivenPositiveLimHitEventIfGlobalResetOrNewMoveReqClearLocalFlags_Test1
VAR_INST
    fbMotionInterlocksLimSw : FB_MotionInterlocksLimSw(
		iMotionInterlocksCommon:=fbMotionInterlocksCommon[1], 
		iLimSwStatus:=fbLimSwStatus[1],
		iMotionLogger := fbMotionLogger[1]
	);
END_VAR
TEST(__POUNAME());
fbLimSwStatus[1].LimitForwardEnable := TRUE;
fbLimSwStatus[1].LimitBackwardEnable := TRUE;
fbMotionInterlocksLimSw.AxisStatus(HomeBusy:=FALSE, PositiveDirection:=TRUE, NegativeDirection:=FALSE);
fbLimSwStatus[1]();
fbMotionInterlocksLimSw();

// Create Forward limit hit event
fbLimSwStatus[1].LimitForwardEnable := FALSE;
fbLimSwStatus[1]();
fbMotionInterlocksLimSw();

// Reset Flags
fbMotionInterlocksLimSw.Reset();
fbMotionInterlocksLimSw();

AssertFalse(Condition := fbMotionInterlocksLimSw.Warning,
               Message := 'Warning should be cleared #1');
AssertFalse(Condition := fbMotionInterlocksLimSw.Warning,
               Message := 'Limit hit flag should be cleared #2');




//Rest axis
fbLimSwStatus[1].LimitForwardEnable := TRUE;
fbLimSwStatus[1].LimitBackwardEnable := TRUE;
fbLimSwStatus[1]();
fbMotionInterlocksLimSw.DriveCommands(MoveEnable:=FALSE, NewMoveReq:=FALSE);
fbMotionInterlocksLimSw.AxisStatus(HomeBusy:=FALSE, PositiveDirection:=FALSE, NegativeDirection:=FALSE);
fbMotionInterlocksLimSw();

// Discrete motion in negative direction
fbMotionInterlocksLimSw.AxisStatus(HomeBusy:=FALSE, PositiveDirection:=FALSE, NegativeDirection:=TRUE);
fbMotionInterlocksLimSw();

// Create backward limit hit event
fbLimSwStatus[1].LimitBackwardEnable := FALSE;
fbLimSwStatus[1]();
fbMotionInterlocksLimSw();

// clear Flags from global reset
fbMotionInterlocksLimSw.Reset();
fbMotionInterlocksLimSw();

AssertFalse(Condition := fbMotionInterlocksLimSw.Warning,
               Message := 'Warning should be cleared #3');
AssertFalse(Condition := fbMotionInterlocksLimSw.Warning,
               Message := 'Limit hit flag should be cleared #4');



//Rest axis
fbLimSwStatus[1].LimitForwardEnable := TRUE;
fbLimSwStatus[1].LimitBackwardEnable := TRUE;
fbLimSwStatus[1]();
fbMotionInterlocksLimSw.DriveCommands(MoveEnable:=FALSE, NewMoveReq:=FALSE);
fbMotionInterlocksLimSw.AxisStatus(HomeBusy:=FALSE, PositiveDirection:=FALSE, NegativeDirection:=FALSE);
fbMotionInterlocksLimSw();

// Discrete motion in positive direction
fbMotionInterlocksLimSw.AxisStatus(HomeBusy:=FALSE, PositiveDirection:=TRUE, NegativeDirection:=FALSE);
fbMotionInterlocksLimSw();

// Create forward limit hit event
fbLimSwStatus[1].LimitForwardEnable := FALSE;
fbLimSwStatus[1]();
fbMotionInterlocksLimSw();

// clear Flags from global reset
fbMotionInterlocksLimSw.DriveCommands(MoveEnable:=FALSE, NewMoveReq:=TRUE);
fbMotionInterlocksLimSw();

AssertFalse(Condition := fbMotionInterlocksLimSw.Warning,
               Message := 'Warning should be cleared #5');
AssertFalse(Condition := fbMotionInterlocksLimSw.Warning,
               Message := 'Limit hit flag should be cleared #6');

TEST_FINISHED();
END_METHOD

END_FUNCTION_BLOCK

// ---- Test/Orchetration/FB_MotionDriveStateMachine_Test.TcPOU
FUNCTION_BLOCK FB_MotionDriveStateMachine_Test EXTENDS FB_TestSuite
VAR
    (*Test all this subject and all dependencies FB_Init call *)


    fbMotionAxisNC : ARRAY [1..20] OF FB_MotionAxisNC_TestDouble;
	stMotionCommand  : ARRAY[1..20] OF ST_MotionCommand;
    fbMotionAxisDS402 : ARRAY [1..8] OF FB_MotionAxisDS402_TestDouble;
    fbMotionLogger : ARRAY [1..20] OF FB_MotionLogger_TestDouble;
    fbMoveRequest : ARRAY [1..20] OF FB_MoveRequest_TestDouble;

END_VAR

GIvenIdlingStateIfErrorGotoErrorState_Test1();
GIvenIdlingStateIfValidatedMoveRequestThenGotoInitState_Test2();
GIvenIdlingStateAndValidatedMoveRequestIfWatchDogTImerOutThenGotoErrorState_Test3();
GivenNCAxisInitStateValidatedAbsoluteMoveRequestThenGotoStartedState_Test4();
GivenNCAxisInitStateValidatedHomeMoveRequestIfModeConfigDoneThenGotoStartedState_Test5();
GivenDS402AxisInitStateValidatedHomeMoveRequestAndNotModeConfigDoneThenLacthInitState_Test15();
GivenDS402AxisInitStateValidatedAbsoluteMoveRequestAndNotModeConfigDoneThenLatchInitState_Test17();
GivenDS402AxisInitStateValidatedHomeMoveRequestAndModeConfigDoneThenGotoStartedState_Test16();
GivenDS402AxisInitStateValidatedAbsoluteMoveRequestAndModeConfigDoneThenGotoStartedState_Test18();
GIvenStartedStatedAndErrorThenGotoErrorState_Test6();
GIvenStartedStateAndBusyStatusFromAxisThenGotoInProgressState_Test7();
GIvenStartedStateAndWatchDogTimeOutThenGotoInProgressState_Test8();
GIvenInPogressStateAndErrorThenGotoErrorState_Test9();
GivenInPogressStateAndAbortedThenGotoInterruptedState_Test10();
GIvenInPogressStateAndHomeMoveDoneStatusFromAxisThenGotoReachedState_Test11();
GIvenInPogressStateAndAbsoluteMoveDoneStatusFromAxisThenGotoReachedState_Test13();
GIvenInterruptedStateAndAbortDoneResetMoveDisablePowerThenGotoIdlingState_Test12();
GIvenReachedStateAndAxisStandStillCompleteMoveRequestThenGotoIdlingState_Test14();

METHOD PRIVATE GivenDS402AxisInitStateValidatedAbsoluteMoveRequestAndModeConfigDoneThenGotoStartedState_Test18
VAR_INST
    fbMotionDriveStateMachine : FB_MotionDriveStateMachine(
		stMotionCommand := THIS^.stMotionCommand[18],
		iMotionAxis:=THIS^.fbMotionAxisDS402[4], 
		iMoveRequest:=THIS^.fbMoveRequest[18],
		iMotionLogger := THIS^.fbMotionLogger[18]
	);
    expectedMoveState : E_MoveState := E_MoveState.STARTED;
    fbTestTimer: TON := (IN:=TRUE, PT:=T#6S);
    nTestStep : INT;
END_VAR
TEST(__POUNAME());
(*DS402 axis modeConfig did not complete within the watchDog timeout*)
CASE nTestStep OF
    0:
        fbMotionDriveStateMachine.State := E_MoveState.IDLING;
        fbMoveRequest[18].Status.bExecute := TRUE;
        fbMoveRequest[18]();
        nTestStep := nTestStep + 1;
    1:
        fbMoveRequest[18].EpicsMotorCommand := E_EpicsMotorCmd.MOVE_ABSOLUTE;
        fbMoveRequest[18]();
        fbMotionAxisDS402[4].ConfigDone := TRUE;
        fbMotionAxisDS402[4]();
        nTestStep := nTestStep + 1;
    2:
        fbMotionDriveStateMachine.State := E_MoveState.INIT;
        nTestStep := nTestStep + 1;
    3:
        AssertEquals_INT(	Expected:=expectedMoveState,
                            Actual:=fbMotionDriveStateMachine.State,
                            Message:='Drive Machine must be in STARTED state #1');
        nTestStep := nTestStep + 1;
        TEST_FINISHED();
END_CASE

fbMotionDriveStateMachine();
fbTestTimer();

IF fbTestTimer.Q THEN
    AssertTrue(Condition := FALSE, Message := CONCAT('Timed out at step: ', TO_STRING(nTestStep)));
    TEST_FINISHED();
END_IF
END_METHOD

METHOD PRIVATE GivenDS402AxisInitStateValidatedAbsoluteMoveRequestAndNotModeConfigDoneThenLatchInitState_Test17
VAR_INST
    fbMotionDriveStateMachine : FB_MotionDriveStateMachine(
		stMotionCommand := THIS^.stMotionCommand[17],
		iMotionAxis:=THIS^.fbMotionAxisDS402[3], 
		iMoveRequest:=THIS^.fbMoveRequest[17],
		iMotionLogger := THIS^.fbMotionLogger[17]
	);
    expectedMoveState : E_MoveState := E_MoveState.INIT;
    fbTestTimer: TON := (IN:=TRUE, PT:=T#6S);
    nTestStep : INT;
END_VAR
TEST(__POUNAME());
(*DS402 axis modeConfig did not complete within the watchDog timeout*)
CASE nTestStep OF
    0:
        fbMotionDriveStateMachine.State := E_MoveState.IDLING;
        fbMoveRequest[17].Status.bExecute := TRUE;
        fbMoveRequest[17]();
        nTestStep := nTestStep + 1;
    1:
        fbMoveRequest[17].EpicsMotorCommand := E_EpicsMotorCmd.MOVE_ABSOLUTE;
        fbMoveRequest[17]();
        fbMotionDriveStateMachine.State := E_MoveState.INIT;
        fbMotionDriveStateMachine();
        nTestStep := nTestStep + 1;
    2:
        AssertEquals_INT(	Expected:=expectedMoveState,
                            Actual:=fbMotionDriveStateMachine.State,
                            Message:='Drive Machine lacthes in INIT state #1');
        nTestStep := nTestStep + 1;
    3:
        IF fbMotionDriveStateMachine.WatchDogTimeOut THEN
            nTestStep := nTestStep + 1;
        END_IF
    4:
        expectedMoveState := E_MoveState.ERROR;
        AssertEquals_INT(	Expected:=expectedMoveState,
                            Actual:=fbMotionDriveStateMachine.State,
                            Message:='Drive Machine lacthes in INIT state #2');
        TEST_FINISHED();
END_CASE

fbMotionDriveStateMachine();
fbTestTimer();

IF fbTestTimer.Q THEN
    AssertTrue(Condition := FALSE, Message := CONCAT('Timed out at step: ', TO_STRING(nTestStep)));
    TEST_FINISHED();
END_IF
END_METHOD

METHOD PRIVATE GivenDS402AxisInitStateValidatedHomeMoveRequestAndModeConfigDoneThenGotoStartedState_Test16
VAR_INST
    fbMotionDriveStateMachine : FB_MotionDriveStateMachine(
		stMotionCommand := THIS^.stMotionCommand[16],
		iMotionAxis:=THIS^.fbMotionAxisDS402[2], 
		iMoveRequest:=THIS^.fbMoveRequest[16],
		iMotionLogger := THIS^.fbMotionLogger[16]
	);
    expectedMoveState : E_MoveState := E_MoveState.STARTED;
    fbTestTimer: TON := (IN:=TRUE, PT:=T#6S);
    nTestStep : INT;
END_VAR
TEST(__POUNAME());
(*DS402 axis modeConfig did not complete within the watchDog timeout*)
CASE nTestStep OF
    0:
        fbMotionDriveStateMachine.State := E_MoveState.IDLING;
        fbMoveRequest[16].Status.bExecute := TRUE;
        fbMoveRequest[16]();
        nTestStep := nTestStep + 1;
    1:
        fbMoveRequest[16].EpicsMotorCommand := E_EpicsMotorCmd.HOME;
        fbMoveRequest[16]();
        fbMotionAxisDS402[2].ConfigDone := TRUE;
        fbMotionAxisDS402[2]();
        nTestStep := nTestStep + 1;
    2:
        fbMotionDriveStateMachine.State := E_MoveState.INIT;
        nTestStep := nTestStep + 1;
    3:
        AssertEquals_INT(	Expected:=expectedMoveState,
                            Actual:=fbMotionDriveStateMachine.State,
                            Message:='Drive Machine must be in STARTED state #1');
        nTestStep := nTestStep + 1;
        TEST_FINISHED();
END_CASE

fbMotionDriveStateMachine();
fbTestTimer();

IF fbTestTimer.Q THEN
    AssertTrue(Condition := FALSE, Message := CONCAT('Timed out at step: ', TO_STRING(nTestStep)));
    TEST_FINISHED();
END_IF
END_METHOD

METHOD PRIVATE GivenDS402AxisInitStateValidatedHomeMoveRequestAndNotModeConfigDoneThenLacthInitState_Test15
VAR_INST
    fbMotionDriveStateMachine : FB_MotionDriveStateMachine(
		stMotionCommand := THIS^.stMotionCommand[15],
		iMotionAxis:=THIS^.fbMotionAxisDS402[1], 
		iMoveRequest:=THIS^.fbMoveRequest[15],
		iMotionLogger := THIS^.fbMotionLogger[15]
	);
    expectedMoveState : E_MoveState := E_MoveState.INIT;
    fbTestTimer: TON := (IN:=TRUE, PT:=T#6S);
    nTestStep : INT;
END_VAR
TEST(__POUNAME());
(*DS402 axis modeConfig did not complete within the watchDog timeout*)
CASE nTestStep OF
    0:
        fbMotionDriveStateMachine.State := E_MoveState.IDLING;
        fbMoveRequest[15].Status.bExecute := TRUE;
        fbMoveRequest[15]();
        nTestStep := nTestStep + 1;
    1:
        fbMoveRequest[15].EpicsMotorCommand := E_EpicsMotorCmd.HOME;
        fbMoveRequest[15]();
        fbMotionDriveStateMachine.State := E_MoveState.INIT;
        fbMotionDriveStateMachine();
        nTestStep := nTestStep + 1;
    2:
        AssertEquals_INT(	Expected:=expectedMoveState,
                            Actual:=fbMotionDriveStateMachine.State,
                            Message:='Drive Machine lacthes in INIT state #1');
        nTestStep := nTestStep + 1;
    3:
        IF fbMotionDriveStateMachine.WatchDogTimeOut THEN
            nTestStep := nTestStep + 1;
        END_IF
    4:
        expectedMoveState := E_MoveState.ERROR;
        AssertEquals_INT(	Expected:=expectedMoveState,
                            Actual:=fbMotionDriveStateMachine.State,
                            Message:='Drive Machine lacthes in INIT state #2');
        TEST_FINISHED();
END_CASE

fbMotionDriveStateMachine();
fbTestTimer();

IF fbTestTimer.Q THEN
    AssertTrue(Condition := FALSE, Message := CONCAT('Timed out at step: ', TO_STRING(nTestStep)));
    TEST_FINISHED();
END_IF
END_METHOD

METHOD PRIVATE GIvenIdlingStateAndValidatedMoveRequestIfWatchDogTImerOutThenGotoErrorState_Test3
VAR_INST
    fbMotionDriveStateMachine : FB_MotionDriveStateMachine(
		stMotionCommand := THIS^.stMotionCommand[3],
		iMotionAxis:=THIS^.fbMotionAxisNC[3], 
		iMoveRequest:=THIS^.fbMoveRequest[3],
		iMotionLogger := THIS^.fbMotionLogger[3]
	);
    expectedMoveState : E_MoveState := E_MoveState.ERROR;
    fbTestTimer: TON := (IN:=TRUE, PT:=T#6S);
    nTestStep : INT;
END_VAR
TEST(__POUNAME());
CASE nTestStep OF
    0:
        fbMotionDriveStateMachine.State := E_MoveState.IDLING;
        fbMoveRequest[3].Status.bExecute := TRUE;
        fbMoveRequest[3]();
        fbMotionDriveStateMachine();
        nTestStep := nTestStep + 1;
    1:
        IF fbMotionDriveStateMachine.WatchDogStatus THEN
            nTestStep := nTestStep + 1;
        END_IF

    2:
        IF fbMotionDriveStateMachine.WatchDogTimeOut THEN
            nTestStep := nTestStep + 1;
        END_IF
    3:
        AssertEquals_INT(	Expected:=expectedMoveState,
                            Actual:=fbMotionDriveStateMachine.State,
                            Message:='Drive Machine state must be ERROR #1');
        AssertTrue(Condition := fbMotionDriveStateMachine.Error, Message := 'Motion Drive state machine must be in error state #2');
        nTestStep := nTestStep + 1;
        TEST_FINISHED();
END_CASE

fbMotionDriveStateMachine();
fbTestTimer();

IF fbTestTimer.Q THEN
    AssertTrue(Condition := FALSE, Message := CONCAT('Timed out at step: ', TO_STRING(nTestStep)));
    TEST_FINISHED();
END_IF
END_METHOD

METHOD PRIVATE GIvenIdlingStateIfErrorGotoErrorState_Test1
VAR_INST
    fbMotionDriveStateMachine : FB_MotionDriveStateMachine(
		stMotionCommand := THIS^.stMotionCommand[1],
		iMotionAxis:=THIS^.fbMotionAxisNC[1], 
		iMoveRequest:=THIS^.fbMoveRequest[1],
		iMotionLogger := THIS^.fbMotionLogger[1]
	);
    expectedMoveState : E_MoveState := E_MoveState.ERROR;
END_VAR
TEST(__POUNAME());

fbMotionDriveStateMachine.State := E_MoveState.IDLING;
fbMotionDriveStateMachine.StateMachine(Error:=TRUE, InterlockEvent:=FALSE);
fbMotionDriveStateMachine();
AssertEquals_INT(	Expected:=expectedMoveState,
                    Actual:=fbMotionDriveStateMachine.State,
                    Message:='Drive Machine state must be ERROR #1');


TEST_FINISHED();
END_METHOD

METHOD PRIVATE GIvenIdlingStateIfValidatedMoveRequestThenGotoInitState_Test2
VAR_INST
    fbMotionDriveStateMachine : FB_MotionDriveStateMachine(
		stMotionCommand := THIS^.stMotionCommand[2],
		iMotionAxis:=THIS^.fbMotionAxisNC[2], 
		iMoveRequest:=THIS^.fbMoveRequest[2],
		iMotionLogger := THIS^.fbMotionLogger[2]
	);
    expectedMoveState : E_MoveState := E_MoveState.INIT;
END_VAR
TEST(__POUNAME());

fbMotionDriveStateMachine.State := E_MoveState.IDLING;
fbMoveRequest[2].Status.bExecute := TRUE;
fbMoveRequest[2]();
fbMotionDriveStateMachine();

AssertEquals_INT(	Expected:=expectedMoveState,
                    Actual:=fbMotionDriveStateMachine.State,
                    Message:='Drive Machine state must be INIT #1');

AssertTrue(Condition := THIS^.fbMoveRequest[2].Status.bExecute, Message := 'Move must be validated #2');

TEST_FINISHED();
END_METHOD

METHOD PRIVATE GivenInPogressStateAndAbortedThenGotoInterruptedState_Test10
VAR_INST
    fbMotionDriveStateMachine : FB_MotionDriveStateMachine(
		stMotionCommand := THIS^.stMotionCommand[10],
		iMotionAxis:=THIS^.fbMotionAxisNC[10], 
		iMoveRequest:=THIS^.fbMoveRequest[10],
		iMotionLogger := THIS^.fbMotionLogger[10]
	);
    expectedMoveState : E_MoveState := E_MoveState.INTERRUPTED;
END_VAR
TEST(__POUNAME());

fbMotionAxisNC[10].Status.bAborted := TRUE;
fbMotionAxisNC[10]();
fbMotionDriveStateMachine.State := E_MoveState.IN_PROGRESS;
fbMotionDriveStateMachine();
AssertEquals_INT(	Expected:=expectedMoveState,
                    Actual:=fbMotionDriveStateMachine.State,
                    Message:='Drive must be in INTERRUPTED state #1');


TEST_FINISHED();
END_METHOD

METHOD PRIVATE GIvenInPogressStateAndAbsoluteMoveDoneStatusFromAxisThenGotoReachedState_Test13
VAR_INST
    fbMotionDriveStateMachine : FB_MotionDriveStateMachine(
		stMotionCommand := THIS^.stMotionCommand[13],
		iMotionAxis:=THIS^.fbMotionAxisNC[13], 
		iMoveRequest:=THIS^.fbMoveRequest[13],
		iMotionLogger := THIS^.fbMotionLogger[13]
	);
    expectedMoveState : E_MoveState := E_MoveState.REACHED;
END_VAR
TEST(__POUNAME());

fbMotionAxisNC[13].Status.bMoveAbsoluteDone := TRUE;
fbMotionAxisNC[13]();
fbMotionDriveStateMachine.State := E_MoveState.IN_PROGRESS;
fbMotionDriveStateMachine();
AssertEquals_INT(	Expected:=expectedMoveState,
                    Actual:=fbMotionDriveStateMachine.State,
                    Message:='Drive must be in REACHED state #1');


TEST_FINISHED();
END_METHOD

METHOD PRIVATE GIvenInPogressStateAndErrorThenGotoErrorState_Test9
VAR_INST
    fbMotionDriveStateMachine : FB_MotionDriveStateMachine(
		stMotionCommand := THIS^.stMotionCommand[9],
		iMotionAxis:=THIS^.fbMotionAxisNC[9], 
		iMoveRequest:=THIS^.fbMoveRequest[9],
		iMotionLogger := THIS^.fbMotionLogger[9]
	);
    expectedMoveState : E_MoveState := E_MoveState.ERROR;
END_VAR
TEST(__POUNAME());

fbMotionDriveStateMachine.State := E_MoveState.IN_PROGRESS;
fbMotionDriveStateMachine.StateMachine(Error:=TRUE, InterlockEvent:=FALSE);
fbMotionDriveStateMachine();

AssertEquals_INT(	Expected:=expectedMoveState,
                    Actual:=fbMotionDriveStateMachine.State,
                    Message:='Drive Machine state must be ERROR #1');

TEST_FINISHED();
END_METHOD

METHOD PRIVATE GIvenInPogressStateAndHomeMoveDoneStatusFromAxisThenGotoReachedState_Test11
VAR_INST
    fbMotionDriveStateMachine : FB_MotionDriveStateMachine(
		stMotionCommand := THIS^.stMotionCommand[11],
		iMotionAxis:=THIS^.fbMotionAxisNC[11], 
		iMoveRequest:=THIS^.fbMoveRequest[11],
		iMotionLogger := THIS^.fbMotionLogger[11]
	);
    expectedMoveState : E_MoveState := E_MoveState.REACHED;
END_VAR
TEST(__POUNAME());

fbMotionAxisNC[11].Status.bHomeDone := TRUE;
fbMotionAxisNC[11]();
fbMotionDriveStateMachine.State := E_MoveState.IN_PROGRESS;
fbMotionDriveStateMachine();
AssertEquals_INT(	Expected:=expectedMoveState,
                    Actual:=fbMotionDriveStateMachine.State,
                    Message:='Drive must be in REACHED state #1');


TEST_FINISHED();
END_METHOD

METHOD PRIVATE GIvenInterruptedStateAndAbortDoneResetMoveDisablePowerThenGotoIdlingState_Test12
VAR_INST
    fbMotionDriveStateMachine : FB_MotionDriveStateMachine(
		stMotionCommand := THIS^.stMotionCommand[12],
		iMotionAxis:=THIS^.fbMotionAxisNC[12], 
		iMoveRequest:=THIS^.fbMoveRequest[12],
		iMotionLogger := THIS^.fbMotionLogger[12]
	);	
    expectedMoveState : E_MoveState := E_MoveState.IDLING;
    fbTestTimer: TON := (IN:=TRUE, PT:=T#2S);
    nTestStep : INT;
END_VAR
TEST(__POUNAME());
CASE 	nTestStep OF
    0:
        fbMotionAxisNC[12].Status.bAborted := TRUE;
        fbMotionDriveStateMachine.State := E_MoveState.IN_PROGRESS;
        nTestStep := nTestStep + 1;
    1:
        // now we should be in the interrupted state
        fbMotionAxisNC[12].Status.bAbortDone := TRUE;
        fbMotionAxisNC[12]();
        nTestStep := nTestStep + 1;
END_CASE

fbMotionAxisNC[12]();
fbMotionDriveStateMachine();
fbTestTimer();

IF nTestStep = 2 THEN
    AssertEquals_INT(	Expected:=expectedMoveState,
                    Actual:=fbMotionDriveStateMachine.State,
                    Message:='Drive must be in IDLING state #1');
    TEST_FINISHED();
ELSIF fbTestTimer.Q THEN
    AssertTrue(Condition := FALSE, Message := CONCAT('Timed out at step: ', TO_STRING(nTestStep)));
    TEST_FINISHED();
END_IF
END_METHOD

METHOD PRIVATE GivenNCAxisInitStateValidatedAbsoluteMoveRequestThenGotoStartedState_Test4
VAR_INST
    fbMotionDriveStateMachine : FB_MotionDriveStateMachine(
		stMotionCommand := THIS^.stMotionCommand[4],
		iMotionAxis:=THIS^.fbMotionAxisNC[4], 
		iMoveRequest:=THIS^.fbMoveRequest[4],
		iMotionLogger := THIS^.fbMotionLogger[4]
	);
    expectedMoveState : E_MoveState := E_MoveState.STARTED;
END_VAR
TEST(__POUNAME());

fbMoveRequest[4].EpicsMotorCommand := E_EpicsMotorCmd.MOVE_ABSOLUTE;
fbMoveRequest[4]();
fbMotionDriveStateMachine.State := E_MoveState.INIT;
fbMotionDriveStateMachine();


expectedMoveState := E_MoveState.STARTED;
AssertEquals_INT(	Expected:=expectedMoveState,
                    Actual:=fbMotionDriveStateMachine.State,
                    Message:='Drive Machine state must be STARTED #1');
TEST_FINISHED();
END_METHOD

METHOD PRIVATE GivenNCAxisInitStateValidatedHomeMoveRequestIfModeConfigDoneThenGotoStartedState_Test5
VAR_INST
    fbMotionDriveStateMachine : FB_MotionDriveStateMachine(
		stMotionCommand := THIS^.stMotionCommand[5],
		iMotionAxis:=THIS^.fbMotionAxisNC[5], 
		iMoveRequest:=THIS^.fbMoveRequest[5],
		iMotionLogger := THIS^.fbMotionLogger[5]
	);
    expectedMoveState : E_MoveState := E_MoveState.ERROR;
    nTestStep : INT;
END_VAR
TEST(__POUNAME());

fbMoveRequest[5].EpicsMotorCommand := E_EpicsMotorCmd.HOME;
fbMoveRequest[5]();
fbMotionDriveStateMachine.State := E_MoveState.INIT;
fbMotionDriveStateMachine();


expectedMoveState := E_MoveState.STARTED;
AssertEquals_INT(	Expected:=expectedMoveState,
                    Actual:=fbMotionDriveStateMachine.State,
                    Message:='Drive Machine state must be STARTED #1');
TEST_FINISHED();
END_METHOD

METHOD PRIVATE GIvenReachedStateAndAxisStandStillCompleteMoveRequestThenGotoIdlingState_Test14
VAR_INST
    fbMotionDriveStateMachine : FB_MotionDriveStateMachine(
		stMotionCommand := THIS^.stMotionCommand[14],
		iMotionAxis:=THIS^.fbMotionAxisNC[14], 
		iMoveRequest:=THIS^.fbMoveRequest[14],
		iMotionLogger := THIS^.fbMotionLogger[14]
	);
    expectedMoveState : E_MoveState := E_MoveState.IDLING;
END_VAR
TEST(__POUNAME());

fbMotionAxisNC[14].Status.bStandStill := TRUE;
fbMotionAxisNC[14].Status.bHomeDone := FALSE;
fbMotionAxisNC[14].Status.bMoveAbsoluteDone := TRUE;
fbMotionAxisNC[14]();
fbMotionDriveStateMachine.State := E_MoveState.REACHED;
fbMotionDriveStateMachine();

AssertEquals_INT(	Expected:=expectedMoveState,
                    Actual:=fbMotionDriveStateMachine.State,
                    Message:='Drive must be in IDLING state #1');


TEST_FINISHED();
END_METHOD

METHOD PRIVATE GIvenStartedStateAndBusyStatusFromAxisThenGotoInProgressState_Test7
VAR_INST
    fbMotionDriveStateMachine : FB_MotionDriveStateMachine(
		stMotionCommand := THIS^.stMotionCommand[7],
		iMotionAxis:=THIS^.fbMotionAxisNC[7], 
		iMoveRequest:=THIS^.fbMoveRequest[7],
		iMotionLogger := THIS^.fbMotionLogger[7]
	);
    expectedMoveState : E_MoveState := E_MoveState.IN_PROGRESS;
    nTestStep : INT;
END_VAR
TEST(__POUNAME());
CASE nTestStep OF
    0:
        fbMotionDriveStateMachine.State := E_MoveState.STARTED;
        fbMotionAxisNC[7].Status.bBusy := TRUE;
        nTestStep := nTestStep + 1;
    1:
        AssertEquals_INT(	Expected:=expectedMoveState,
                            Actual:=fbMotionDriveStateMachine.State,
                            Message:='Drive Machine must be IN_PROGRESS state #1');
        TEST_FINISHED();
END_CASE

fbMotionDriveStateMachine();
END_METHOD

METHOD PRIVATE GIvenStartedStateAndWatchDogTimeOutThenGotoInProgressState_Test8
VAR_INST
    fbMotionDriveStateMachine : FB_MotionDriveStateMachine(
		stMotionCommand := THIS^.stMotionCommand[8],
		iMotionAxis:=THIS^.fbMotionAxisNC[8], 
		iMoveRequest:=THIS^.fbMoveRequest[8],
		iMotionLogger := THIS^.fbMotionLogger[8]
	);
    expectedMoveState : E_MoveState := E_MoveState.ERROR;
    fbTestTimer: TON := (IN:=TRUE, PT:=T#6S);
    nTestStep : INT;
END_VAR
TEST(__POUNAME());
CASE nTestStep OF
    0:
        fbMoveRequest[8].Status.bExecute := TRUE;
        fbMoveRequest[8]();
        fbMotionDriveStateMachine.State := E_MoveState.STARTED;
        fbMotionDriveStateMachine.WatchDog := TRUE;
        fbMotionDriveStateMachine();
        nTestStep := nTestStep + 1;
    1:
        IF fbMotionDriveStateMachine.WatchDogStatus THEN
            nTestStep := nTestStep + 1;
        END_IF

    2:
        IF fbMotionDriveStateMachine.WatchDogTimeOut THEN
            nTestStep := nTestStep + 1;
        END_IF
    3:
        AssertEquals_INT(	Expected:=expectedMoveState,
                            Actual:=fbMotionDriveStateMachine.State,
                            Message:='Drive Machine state must be ERROR #1');
        AssertTrue(Condition := fbMotionDriveStateMachine.Error, Message := 'Motion Drive state machine must be in error state #2');
        nTestStep := nTestStep + 1;
        TEST_FINISHED();
END_CASE

fbMotionDriveStateMachine();
fbTestTimer();

IF fbTestTimer.Q THEN
    AssertTrue(Condition := FALSE, Message := CONCAT('Timed out at step: ', TO_STRING(nTestStep)));
    TEST_FINISHED();
END_IF
END_METHOD

METHOD PRIVATE GIvenStartedStatedAndErrorThenGotoErrorState_Test6
VAR_INST
    fbMotionDriveStateMachine : FB_MotionDriveStateMachine(
		stMotionCommand := THIS^.stMotionCommand[6],
		iMotionAxis:=THIS^.fbMotionAxisNC[6], 
		iMoveRequest:=THIS^.fbMoveRequest[6],
		iMotionLogger := THIS^.fbMotionLogger[6]
	);
    expectedMoveState : E_MoveState := E_MoveState.ERROR;

    nTestStep : INT;
END_VAR
TEST(__POUNAME());
CASE nTestStep OF
    0:
        fbMotionDriveStateMachine.State := E_MoveState.STARTED;
        fbMotionDriveStateMachine.StateMachine(Error:=TRUE, InterlockEvent:=FALSE);
        nTestStep := nTestStep + 1;
    1:
        AssertEquals_INT(	Expected:=expectedMoveState,
                            Actual:=fbMotionDriveStateMachine.State,
                            Message:='Drive Machine must be ERROR state #1');
        TEST_FINISHED();
END_CASE

fbMotionDriveStateMachine();
END_METHOD

END_FUNCTION_BLOCK

// ---- Test/TestDouble/FB_MotionAxisDS402_TestDouble.TcPOU
FUNCTION_BLOCK FB_MotionAxisDS402_TestDouble IMPLEMENTS I_MotionAxisDS402
VAR
    bError: BOOL;
    nErrorID: UDINT;
    sMessage : T_MAXSTRING;
    stMotionAxisStatus : ST_AxisStatus;
    bConfigDone : BOOL;
END_VAR

METHOD AxisEnabled : BOOL
END_METHOD

(*
    Handle positive/negative backlash compensation
    User needs to set the direction of backlash from the sign of the compensation value
    Backlash compensation is disabled during referencing (homing).
    When direction is positive/negative, further movement in the negative/positive direction not compensated
    further movement in the negative/positive direction will be compensated
*)
METHOD BacklashCompensation
VAR_INPUT
    Enable	: BOOL := FALSE;
    RampVelo	: LREAL;
END_VAR
END_METHOD

METHOD ClearHaltStatus
END_METHOD

{warning 'Add method implementation '}
METHOD ClearHomeStatus
END_METHOD

{warning 'Add method implementation '}
METHOD ClearMoveAbsoluteStatus
END_METHOD

METHOD ClearResetStatus
END_METHOD

PROPERTY ConfigDone : BOOL
GET
ConfigDone := bConfigDone;
END_GET
SET
bConfigDone := ConfigDone;
END_SET
END_PROPERTY

METHOD DisablePower
END_METHOD

METHOD DriveCommands
VAR_INPUT
    HomeCmd	: BOOL;
    NewMoveReq	: BOOL;
    EnableMode	: E_StageEnableMode;
END_VAR
END_METHOD

METHOD Halt
VAR_INPUT
    Deceleration	: LREAL := 0;
    Jerk	: LREAL := 0;
    BufferMode	: MC_BufferMode := MC_BufferMode.MC_Aborting;
END_VAR
END_METHOD

METHOD Home
VAR_INPUT
    Position        : LREAL         := DEFAULT_HOME_POSITION;
    BufferMode      : MC_BufferMode;
 	HomeMode: INT :=E_EpicsHomeCmd.NONE;
END_VAR
END_METHOD

{warning 'Add method implementation '}
METHOD HomeAbortRecovery
END_METHOD

METHOD ModeConfigDone : BOOL
VAR_INPUT
    Mode	: E_EpicsMotorCmd;
END_VAR
 ModeConfigDone :=  bConfigDone;
END_METHOD

METHOD ModeOfOperation : BOOL
VAR_INPUT
    RecentModeOfOperation	: E_DS402OpMode;
END_VAR
END_METHOD

METHOD MoveAbsolute
VAR_INPUT
    Position	: LREAL;
    Velocity	: LREAL;
    Acceleration	: LREAL := 0;
    Deceleration	: LREAL := 0;
    Jerk	: LREAL := 0;
    BufferMode	: MC_BufferMode := MC_BufferMode.MC_Aborting;
END_VAR
END_METHOD

METHOD Power
VAR_INPUT
    Enable	: BOOL;
    Enable_Positive	: BOOL;
    Enable_Negative	: BOOL;
    Override	: LREAL;
    BufferMode	: MC_BufferMode;
END_VAR
END_METHOD

METHOD ReadAxisParams
VAR_INPUT
    Enable	: BOOL;
    RefreshDelay	: TIME;
END_VAR
END_METHOD

METHOD Reset
END_METHOD

METHOD SaveAxisParams
VAR_INPUT
    Enable	: BOOL;
END_VAR
END_METHOD

PROPERTY Status : REFERENCE TO ST_AxisStatus
GET
Status REF= stMotionAxisStatus;
END_GET
END_PROPERTY

END_FUNCTION_BLOCK

// ---- Test/Orchetration/FB_MoveRequest_Test.TcPOU
FUNCTION_BLOCK FB_MoveRequest_Test EXTENDS FB_TestSuite
VAR
        stMotionCommand :  ARRAY[1..10] OF ST_MotionCommand;
		stMotionStatus :  ARRAY[1..10] OF ST_MotionStatus;
END_VAR

GivenMoveRequestAndInterlockAndErrorStatusUpdateRequestStatus_Test1();
GivenMoveRequestDisabledWhenInterlockFalseAlwaysMode_Test2();
GivenAlwaysModeEnableWhenInterlockTrue_Test3();
GivenDuringMotionDisableWhenInterlockFalse_Test4();
GivenDuringMotionEnableWhenInterlockTrue_Test5();
GivenAbsoluteMoveCorrectFlags_Test6();
GivenHomeMoveCorrectFlags_Test7();
GivenInitMoveRequestSetsBusyClearsDoneAndErrorMsg_Test8();
GivenExecuteFlagsSetAndCleared_Test9();

METHOD PRIVATE GivenAbsoluteMoveCorrectFlags_Test6
VAR_INST
    fbMoveRequest : FB_EpicsMoveRequest(
		stMotionCommand:=stMotionCommand[7],
		stMotionStatus:=stMotionStatus[7]
	);
	eExpectedMoveMode :E_EpicsMotorCmd := E_EpicsMotorCmd.MOVE_ABSOLUTE;
END_VAR
// ----------- Absolute Move Command: flags and mode correctness -------------
TEST(__POUNAME());

fbMoveRequest.MoveRequestCmds(
    HomeCmd    := FALSE,
    MoveCmd    := TRUE,
    MoveOk     := TRUE,
    EnableDone := TRUE,
    HomeMode   := E_EpicsHomeCmd.NONE,
    EnableMode := E_StageEnableMode.DURING_MOTION
);
fbMoveRequest();

AssertTrue(fbMoveRequest.Status.bNewMoveReq, 'Should register move request');
AssertTrue(fbMoveRequest.Status.bExecMove, 'Should be ready for move');
AssertFalse(fbMoveRequest.Status.bExecHome, 'Should not be ready for home');
AssertEquals_INT(eExpectedMoveMode, fbMoveRequest.Status.nCommand, 'Command=absolute');
TEST_FINISHED();
END_METHOD

METHOD PRIVATE GivenAlwaysModeEnableWhenInterlockTrue_Test3
VAR_INST
    fbMoveRequest : FB_EpicsMoveRequest(
		stMotionCommand:=stMotionCommand[4],
		stMotionStatus:=stMotionStatus[4]
	);
END_VAR
// ----------- Always mode: should enable if interlock met -------------
TEST(__POUNAME());

fbMoveRequest.MoveRequestCmds(
    HomeCmd    := FALSE,
    MoveCmd    := TRUE,
    MoveOk     := TRUE,
    EnableDone := TRUE,
    HomeMode   := E_EpicsHomeCmd.NONE,
    EnableMode := E_StageEnableMode.ALWAYS
);
fbMoveRequest();

AssertTrue( fbMoveRequest.Status.bEnable, 'Should be enabled when MoveOk is TRUE in ALWAYS mode' );
TEST_FINISHED();
END_METHOD

METHOD PRIVATE GivenDuringMotionDisableWhenInterlockFalse_Test4
VAR_INST
    fbMoveRequest : FB_EpicsMoveRequest(
		stMotionCommand:=stMotionCommand[5],
		stMotionStatus:=stMotionStatus[5]
	);
END_VAR
// ----------- DuringMotion: Must not enable if interlock not met -------------
TEST(__POUNAME());
fbMoveRequest.MoveRequestCmds(
    HomeCmd    := FALSE,
    MoveCmd    := TRUE,
    MoveOk     := FALSE,
    EnableDone := TRUE,
    HomeMode   := E_EpicsHomeCmd.NONE,
    EnableMode := E_StageEnableMode.DURING_MOTION
);
fbMoveRequest();

AssertFalse(fbMoveRequest.Status.bEnable, 'Request disabled if MoveOk is FALSE in DURING_MOTION mode');
TEST_FINISHED();
END_METHOD

METHOD PRIVATE GivenDuringMotionEnableWhenInterlockTrue_Test5
VAR_INST
    fbMoveRequest : FB_EpicsMoveRequest(
		stMotionCommand:=stMotionCommand[6],
		stMotionStatus:=stMotionStatus[6]
	);
END_VAR
TEST(__POUNAME());

fbMoveRequest.MoveRequestCmds(
    HomeCmd    := FALSE,
    MoveCmd    := TRUE,
    MoveOk     := TRUE,
    EnableDone := TRUE,
    HomeMode   := E_EpicsHomeCmd.NONE,
    EnableMode := E_StageEnableMode.DURING_MOTION
);
fbMoveRequest();

AssertTrue(fbMoveRequest.Status.bEnable, 'Request enabled when MoveOk TRUE in DURING_MOTION mode');
TEST_FINISHED();
END_METHOD

METHOD PRIVATE GivenExecuteFlagsSetAndCleared_Test9
VAR_INST
    fbMoveRequest : FB_EpicsMoveRequest(
		stMotionCommand:=stMotionCommand[10],
		stMotionStatus:=stMotionStatus[10]
	);
END_VAR
// ----------- Execute flags set and cleared as expected -------------
TEST(__POUNAME());

	fbMoveRequest.MoveRequestCmds(
		HomeCmd    := FALSE,
		MoveCmd    := TRUE,
		MoveOk     := TRUE,
		EnableDone := TRUE,
		HomeMode   := E_EpicsHomeCmd.NONE,
		EnableMode := E_StageEnableMode.DURING_MOTION
	);
	fbMoveRequest();
	
	AssertTrue(fbMoveRequest.stMotionRequestStatus.bExecute, 'bExecute must be set');
	AssertTrue(fbMoveRequest.Status.bExecute, 'Local execute flag must be set');
	
	// Simulate user reset/stop
	fbMoveRequest.StopMoveRequest();
	fbMoveRequest();
	AssertTrue(fbMoveRequest.Status.bPrepareDisable, 'Request must prepare disable after clear');

TEST_FINISHED();
END_METHOD

METHOD PRIVATE GivenHomeMoveCorrectFlags_Test7
VAR_INST
    fbMoveRequest : FB_EpicsMoveRequest(
		stMotionCommand:=stMotionCommand[8],
		stMotionStatus:=stMotionStatus[8]
	);
	nActualMoveMode : INT;
	eExpectedMoveMode :E_EpicsMotorCmd := E_EpicsMotorCmd.HOME;
END_VAR
// ----------- Home Move Command: flags and mode correctness -------------
TEST(__POUNAME());

	fbMoveRequest.MoveRequestCmds(
		HomeCmd    := TRUE,
		MoveCmd    := FALSE,
		MoveOk     := TRUE,
		EnableDone := TRUE,
		HomeMode   := E_EpicsHomeCmd.LOW_LIMIT,
		EnableMode := E_StageEnableMode.DURING_MOTION
	);
	fbMoveRequest();
	
	nActualMoveMode := fbMoveRequest.Status.nCommand;
	AssertTrue(fbMoveRequest.Status.bNewMoveReq, 'Registered home request');
	AssertFalse(fbMoveRequest.Status.bExecMove, 'Should not be absolute for home');
	AssertTrue(fbMoveRequest.Status.bExecHome, 'Home move must be ready');
	AssertEquals_INT(eExpectedMoveMode, nActualMoveMode, 'Command=home');
TEST_FINISHED();
END_METHOD

METHOD PRIVATE GivenInitMoveRequestSetsBusyClearsDoneAndErrorMsg_Test8
VAR_INST
    fbMoveRequest : FB_EpicsMoveRequest(
		stMotionCommand:=stMotionCommand[9],
		stMotionStatus:=stMotionStatus[9]
	);
	sMoveMessage : STRING := '';
END_VAR
// ----------- Init should set busy, clear done, clear error string -------------
TEST(__POUNAME());

	fbMoveRequest.MoveRequestCmds(
		HomeCmd    := FALSE,
		MoveCmd    := TRUE,
		MoveOk     := TRUE,
		EnableDone := TRUE,
		HomeMode   := E_EpicsHomeCmd.NONE,
		EnableMode := E_StageEnableMode.DURING_MOTION
	);

	fbMoveRequest.InitMoveRequest();
	fbMoveRequest();
	
	AssertTrue(stMotionStatus[9].bBusy, 'Busy at init');
	AssertFalse(stMotionStatus[9].bDone, 'Done reset at init');
	AssertEquals_STRING(sMoveMessage, stMotionStatus[9].sErrorMessage, 'Error cleared at init');
TEST_FINISHED();
END_METHOD

METHOD PRIVATE GivenMoveRequestAndInterlockAndErrorStatusUpdateRequestStatus_Test1
VAR_INST
    fbMoveRequest : FB_EpicsMoveRequest(stMotionCommand:=stMotionCommand[1], stMotionStatus:=stMotionStatus[1]);
    eExpectedMoveMode : INT := E_EpicsMotorCmd.MOVE_ABSOLUTE;
    eActualMoveMode : INT;
    sMoveMessage : STRING := '';
END_VAR
TEST(__POUNAME());

	// ------------------------
	// ALWAYS mode: request should only enable when allowed, and latch off on error
	// ------------------------
	fbMoveRequest.MoveRequestCmds(
		HomeCmd := FALSE,
		MoveCmd := FALSE,
		MoveOk := FALSE,
		EnableDone := FALSE,
		HomeMode := E_EpicsHomeCmd.NONE,
		EnableMode := E_StageEnableMode.ALWAYS
	);
	fbMoveRequest();
	
	AssertFalse(
		fbMoveRequest.Status.bEnable,
		'move request must be disabled with invalid interlock in ALWAYS mode #1'
	);
	
	fbMoveRequest.MoveRequestCmds(
		HomeCmd := FALSE,
		MoveCmd := TRUE,
		MoveOk := TRUE,
		EnableDone := TRUE,
		HomeMode := E_EpicsHomeCmd.NONE,
		EnableMode := E_StageEnableMode.ALWAYS
	);
	fbMoveRequest();
	
	AssertTrue(
		fbMoveRequest.Status.bEnable,
		'move request must be enabled with valid interlock in ALWAYS mode #2'
	);
	
	// Now simulate a persistent/latching error after enable
	fbMoveRequest.ClearMoveRequest();
	fbMoveRequest();
	
	stMotionstatus[1].bError := TRUE; // Simulate latching error
	fbMoveRequest.MoveRequestCmds(
		HomeCmd := FALSE,
		MoveCmd := TRUE,
		MoveOk := TRUE,
		EnableDone := TRUE,
		HomeMode := E_EpicsHomeCmd.NONE,
		EnableMode := E_StageEnableMode.ALWAYS
	);
	fbMoveRequest();
	
	AssertFalse(
		fbMoveRequest.Status.bEnable,
		'Latching error condition must disable move request in ALWAYS mode #3'
	);
	
	// ------------------------
	// DURING_MOTION mode: only enable when MoveOk, must stay off with error or missing enables
	// ------------------------
	// 
	// Clear previous request
	fbMoveRequest.ClearMoveRequest();
	fbMoveRequest.ClearMoveRequestErrors();
	fbMoveRequest();
	
	fbMoveRequest.MoveRequestCmds(
		HomeCmd := FALSE,
		MoveCmd := TRUE,
		MoveOk := FALSE,
		EnableDone := FALSE,
		HomeMode := E_EpicsHomeCmd.NONE,
		EnableMode := E_StageEnableMode.DURING_MOTION
	);
	fbMoveRequest();
	
	AssertFalse(
		fbMoveRequest.Status.bEnable,
		'Missing MoveOk must keep move disabled in DURING_MOTION mode #4'
	);
	
	fbMoveRequest.ClearMoveRequest();
	fbMoveRequest();
	
	fbMoveRequest.MoveRequestCmds(
		HomeCmd := FALSE,
		MoveCmd := TRUE,
		MoveOk := TRUE,
		EnableDone := FALSE,
		HomeMode := E_EpicsHomeCmd.NONE,
		EnableMode := E_StageEnableMode.DURING_MOTION
	);
	fbMoveRequest();
	
	AssertTrue(
		fbMoveRequest.Status.bEnable,
		'Move request must be enabled in DURING_MOTION mode #6'
	);
	
	fbMoveRequest.ClearMoveRequest();
	fbMoveRequest();
	
	fbMoveRequest.MoveRequestCmds(
		HomeCmd := FALSE,
		MoveCmd := TRUE,
		MoveOk := TRUE,
		EnableDone := TRUE,
		HomeMode := E_EpicsHomeCmd.NONE,
		EnableMode := E_StageEnableMode.DURING_MOTION
	);
	fbMoveRequest();
	
	eExpectedMoveMode := E_EpicsMotorCmd.MOVE_ABSOLUTE;
	
	AssertTrue(fbMoveRequest.Status.bNewMoveReq, 'Move request must be Registered #7');
	AssertTrue(fbMoveRequest.Status.bExecMove, 'Absolute move must be ready #8');
	AssertFalse(fbMoveRequest.Status.bExecHome, 'Move is not a Homing move #9');
	AssertEquals_INT(eExpectedMoveMode, fbMoveRequest.Status.nCommand, 'Move command must be absolute #10');
	
	fbMoveRequest.ClearMoveRequest();
	fbMoveRequest();
	
	fbMoveRequest.MoveRequestCmds(
		HomeCmd := TRUE,
		MoveCmd := FALSE,
		MoveOk := TRUE,
		EnableDone := TRUE,
		HomeMode := E_EpicsHomeCmd.LOW_LIMIT,
		EnableMode := E_StageEnableMode.DURING_MOTION
	);
	fbMoveRequest();
	
	eExpectedMoveMode := E_EpicsMotorCmd.HOME;
	eActualMoveMode := fbMoveRequest.Status.nCommand;
	
	AssertTrue(fbMoveRequest.Status.bNewMoveReq, 'Move request must be Registered #11');
	AssertFalse(fbMoveRequest.Status.bExecMove, 'Move is not Absolute #12');
	AssertTrue(fbMoveRequest.Status.bExecHome, 'Home move must be ready #13');
	AssertEquals_INT(eExpectedMoveMode, eActualMoveMode, 'Move command must be a valid homing mode #14');
	
	fbMoveRequest.ClearMoveRequest();
	fbMoveRequest();
	
	stMotionstatus[1].bError := FALSE;
	fbMoveRequest.MoveRequestCmds(
		HomeCmd := FALSE,
		MoveCmd := TRUE,
		MoveOk := TRUE,
		EnableDone := TRUE,
		HomeMode := E_EpicsHomeCmd.NONE,
		EnableMode := E_StageEnableMode.DURING_MOTION
	);
	fbMoveRequest.InitMoveRequest();
	fbMoveRequest();
	
	AssertTrue(stMotionstatus[1].bBusy, 'Move Request Busy flag must be set at init #15');
	AssertFalse(stMotionstatus[1].bDone, 'Move request Done flag must reset at init #16');
	AssertEquals_STRING(sMoveMessage, stMotionstatus[1].sErrorMessage, 'Move request Error flag must be cleared at init #17');
	
	fbMoveRequest.ClearMoveRequest();
	fbMoveRequest();
	
	stMotionstatus[1].bError := FALSE;
	fbMoveRequest.MoveRequestCmds(
		HomeCmd := FALSE,
		MoveCmd := TRUE,
		MoveOk := TRUE,
		EnableDone := TRUE,
		HomeMode := E_EpicsHomeCmd.NONE,
		EnableMode := E_StageEnableMode.DURING_MOTION
	);
	fbMoveRequest();
	
	AssertTrue(fbMoveRequest.stMotionRequestStatus.bExecute, 'Execute must be set by now #18');
	AssertTrue(fbMoveRequest.Status.bExecute, 'Local Execute must be set by now #19');
	
	// Simulate user stop
	fbMoveRequest.StopMoveRequest();
	fbMoveRequest();
	
	AssertTrue(fbMoveRequest.Status.bPrepareDisable, 'Must be preparing to disable by now #20');

TEST_FINISHED();
END_METHOD

METHOD PRIVATE GivenMoveRequestDisabledWhenInterlockFalseAlwaysMode_Test2
VAR_INST
    fbMoveRequest : FB_EpicsMoveRequest(
		stMotionCommand:=stMotionCommand[3],
		stMotionStatus:=stMotionStatus[3]
	);
END_VAR
// ----------- Always mode: should NOT enable if interlock not met -------------
TEST(__POUNAME());
	
	fbMoveRequest.MoveRequestCmds(
		HomeCmd    := FALSE,
		MoveCmd    := FALSE,
		MoveOk     := FALSE,
		EnableDone := FALSE,
		HomeMode   := E_EpicsHomeCmd.NONE,
		EnableMode := E_StageEnableMode.ALWAYS
	);
	fbMoveRequest();
	
	AssertFalse(fbMoveRequest.Status.bEnable, 'Should be disabled if MoveOk is FALSE in ALWAYS mode');
TEST_FINISHED();
END_METHOD

END_FUNCTION_BLOCK

// ---- Test/NC/FB_NcMotionBlocks_Test.TcPOU
FUNCTION_BLOCK FB_NcMotionBlocks_Test EXTENDS FB_TestSuite
VAR
    fbAxisRef : ARRAY [1..16] OF AXIS_REF;
    fbLimSwStatus : ARRAY [1..16] OF FB_LimSwStatus_TestDouble;
    fbMotionLogger : ARRAY [1..16] OF FB_MotionLogger_TestDouble;
    fbPower : ARRAY [1..16] OF FB_PowerNC[	(AxisRef := fbAxisRef[1], iMotionLogger:= fbMotionLogger[1]),
                                            (AxisRef := fbAxisRef[2], iMotionLogger:= fbMotionLogger[2]),
                                            (AxisRef := fbAxisRef[3], iMotionLogger:= fbMotionLogger[3]),
                                            (AxisRef := fbAxisRef[4], iMotionLogger:= fbMotionLogger[4]),
                                            (AxisRef := fbAxisRef[5], iMotionLogger:= fbMotionLogger[5]),
                                            (AxisRef := fbAxisRef[6], iMotionLogger:= fbMotionLogger[6]),
                                            (AxisRef := fbAxisRef[7], iMotionLogger:= fbMotionLogger[7]),
                                            (AxisRef := fbAxisRef[8], iMotionLogger:= fbMotionLogger[8]),
											(AxisRef := fbAxisRef[9], iMotionLogger:= fbMotionLogger[9]),
                                            (AxisRef := fbAxisRef[10], iMotionLogger:= fbMotionLogger[10]),
                                            (AxisRef := fbAxisRef[11], iMotionLogger:= fbMotionLogger[11]),
                                            (AxisRef := fbAxisRef[12], iMotionLogger:= fbMotionLogger[12]),
                                            (AxisRef := fbAxisRef[13], iMotionLogger:= fbMotionLogger[13]),
                                            (AxisRef := fbAxisRef[14], iMotionLogger:= fbMotionLogger[14]),
                                            (AxisRef := fbAxisRef[15], iMotionLogger:= fbMotionLogger[15]),
                                            (AxisRef := fbAxisRef[16], iMotionLogger:= fbMotionLogger[16])
                                            ];
END_VAR

GivenHomeCmdAbsoluteSetModeThenSetHomeDoneAndPositionToUserDefineOffset_Test1();
GivenHomeCmdBacklashCompensationInactiveThenMoveStartandCompletesWithBacklashCompensationDisabled_Test2();
GivenHomeCmdHomeViaHighModeAndHomeSwPulseThenMoveToUserDefineOffset_Test3();
GivenHomeCmdHomeViaHighModeForwardSwPulseBeforeHomeSwPulseThenMoveToUserDefineOffset_Test4();
GivenHomeCmdHomeViaLowModeAndHomeSwPulseThenMoveToUserDefineOffset_Test5();
GivenHomeCmdHomeViaLowModeBackwardSwPulseBeforeHomeSwPulseThenMoveToUserDefineOffset_Test6();
GivenHomeCmdLowLimitModeAndABackwardSwPulseThenHomeDoneAndPositionSetToUserDefineOffset_Test7();
GivenHomeCmdNoneModeThenSetHomeFlag_Test8();
GivenHomeCmdSetToHighLimitAndHighLimitPulseThenSetHomeDoneAndPositionToUserDefineOffset_Test9();
GivenMoveCmdNegativeBacklashCompensationActiveThenReverseMoveIsCompensated_Test10();
GivenMoveCmdPositiveBacklashCompensationActiveThenReverseMoveIsCompensated_Test11();
GivenDirectionalPowerEnabledAndBackwardAbsoluteMoveIfNegativeLimitHitThenAbortMove_Test12();
GivenDirectionalPowerEnabledAndForwardAbsoluteMoveIfPositiveLimitHitThenAbortMove_Test13();
GivenPowerIsEnabledAndCompletedAbsoluteMoveThenMoveAbsoluteDoneStatusRetained_Test14();
GivenPowerIsEnabledAndAbsoluteMoveStartedIfHaltSignalThenMoveIsAbortedAndHaltDoneIsRetained_Test15();
GivenPowerIsEnabledAbsoluteMoveIfResetThenMoveIsAbortedAndResetDoneIsRetained_Test16();

//

METHOD PRIVATE GivenDirectionalPowerEnabledAndBackwardAbsoluteMoveIfNegativeLimitHitThenAbortMove_Test12
VAR_INST
    // Subject under tests
    fbMoveAbsolute : FB_MoveAbsoluteNC(AxisRef := fbAxisRef[12],  iMotionLogger:= fbMotionLogger[12]);
    fbTestTimer : TON := (PT := T#3S, IN := TRUE);
    nTestStateStep : INT;
    fbLimtHitTimer : TON := (PT := T#1S, IN := FALSE);
    fExpectedPosition: LREAL := 50.0;
END_VAR
TEST(__POUNAME());

// Cyclically call these every scan for correct PLC logic
fbPower[12].Power(
    Enable := TRUE,
    Enable_Positive := fbLimSwStatus[12].LimitForwardEnable,
    Enable_Negative := fbLimSwStatus[12].LimitBackwardEnable,
    Override := 100
);

// Stepwise state machine logic
CASE nTestStateStep OF
    0 : // Wait for power on before initiating move
        IF fbPower[12].PowerIsEnabled THEN
            nTestStateStep := 1;
        END_IF

    1 : // Issue negative move and start timer
        fbMoveAbsolute.MoveAbsolute(
            Position := -150.0,
            Velocity := 100,
            Acceleration := 200,
            Deceleration := 200
        );
        fbLimtHitTimer.IN := TRUE;
        nTestStateStep := 2;

    2 : // After timer, simulate limit hit
        IF fbLimtHitTimer.Q THEN
            fbLimSwStatus[12].LimitBackwardEnable := FALSE; // Simulate the axis hitting the negative limit
            nTestStateStep := 3;
        END_IF

    3 : // Wait until move is aborted by limit hit
        IF fbMoveAbsolute.Aborted THEN
            nTestStateStep := 4;
        END_IF

    4 : // Assertions below once test finished
END_CASE

// Cyclic calls required for correct behavior
fbLimtHitTimer();
fbTestTimer();
fbAxisRef[12].ReadStatus();
fbMoveAbsolute();

// Final assertion and test finish
IF nTestStateStep = 4 THEN
    AssertTrue(
        Condition := fbAxisRef[12].Status.HasBeenStopped,
        Message := 'Expected HasBeenStopped after move aborted by limit'
    );
    TEST_FINISHED();

ELSIF fbTestTimer.Q THEN
    AssertTrue(
        Condition := FALSE,
        Message := CONCAT('Timed out at step: ', TO_STRING(nTestStateStep))
    );
    TEST_FINISHED();
END_IF
END_METHOD

METHOD PRIVATE GivenDirectionalPowerEnabledAndForwardAbsoluteMoveIfPositiveLimitHitThenAbortMove_Test13
VAR_INST

    // Subject under tests
    fbMoveAbsolute : FB_MoveAbsoluteNC(AxisRef := fbAxisRef[13], iMotionLogger:= fbMotionLogger[13]);
    fbTestTimer : TON := (PT := T#3S, IN := TRUE);
    nTestStateStep : INT;
    fbLimtHitTimer : TON := (PT := T#1S, IN := FALSE);
    fExpectedPosition: LREAL := 50.0;
END_VAR
TEST(__POUNAME());

// Cyclically call these every scan for correct PLC logic
fbPower[13].Power(
    Enable := TRUE,
    Enable_Positive := fbLimSwStatus[13].LimitForwardEnable,
    Enable_Negative := fbLimSwStatus[13].LimitBackwardEnable,
    Override := 100
);

// Stepwise state machine logic
CASE nTestStateStep OF
    0 : // Wait for power on before initiating move
        IF fbPower[13].PowerIsEnabled THEN
            nTestStateStep := 1;
        END_IF

    1 : // Issue negative move and start timer
        fbMoveAbsolute.MoveAbsolute(
            Position := 150.0,
            Velocity := 100,
            Acceleration := 200,
            Deceleration := 200
        );
        fbLimtHitTimer.IN := TRUE;
        nTestStateStep := 2;

    2 : // After timer, simulate limit hit
        IF fbLimtHitTimer.Q THEN
            fbLimSwStatus[13].LimitForwardEnable := FALSE; // Simulate the axis hitting the negative limit
            nTestStateStep := 3;
        END_IF

    3 : // Wait until move is aborted by limit hit
        IF fbMoveAbsolute.Aborted THEN
            nTestStateStep := 4;
        END_IF
END_CASE

// Cyclic calls required for correct behavior
fbLimtHitTimer();
fbTestTimer();
fbAxisRef[13].ReadStatus();
fbMoveAbsolute();

// Final assertion and test finish
IF nTestStateStep = 4 THEN
    AssertTrue(
        Condition := fbAxisRef[13].Status.HasBeenStopped,
        Message := 'Expected HasBeenStopped after move aborted by limit'
    );
    TEST_FINISHED();

ELSIF fbTestTimer.Q THEN
    AssertTrue(
        Condition := FALSE,
        Message := CONCAT('Timed out at step: ', TO_STRING(nTestStateStep))
    );
    TEST_FINISHED();
END_IF
END_METHOD

METHOD PRIVATE GivenHomeCmdAbsoluteSetModeThenSetHomeDoneAndPositionToUserDefineOffset_Test1
VAR_INST
	// 
    fbHome : FB_HomeNC(
		AxisRef:=fbAxisRef[1],
		iLimSwStatus:=fbLimSwStatus[1],
		iMotionLogger:=fbMotionLogger[1]
	)	:=	(	Mode:=E_EpicsHomeCmd.ABSOLUTE_SET	);

    fbTestTimer : TON := (IN := TRUE, PT := T#8S);
    nTestStep : INT := 0;
    fExpectedPosition : LREAL := 20.0;
    fActPosition : LREAL := 0.0;
    bCalibrated : BOOL := FALSE;
END_VAR
TEST(__POUNAME());
// FBs that must be invoked cyclically
fbLimSwStatus[1]();
fbMotionLogger[1]();
fbAxisRef[1].ReadStatus();
fbPower[1].Power(
    Enable := TRUE,
    Enable_Positive := fbLimSwStatus[1].LimitForwardEnable,
    Enable_Negative := fbLimSwStatus[1].LimitBackwardEnable,
    Override := 100.0
);
fbHome();
fbTestTimer(IN := TRUE);

// --- State Machine ---
CASE nTestStep OF
    0: // Enable power, then issue home command
        IF fbPower[1].PowerIsEnabled THEN
            fbHome.Home(
				Position := fExpectedPosition,
				BufferMode := MC_BufferMode.MC_Aborting,
				HomeMode:=E_EpicsHomeCmd.ABSOLUTE_SET
			);
            nTestStep := 1;
        END_IF

    1: // Wait for homing to complete
        IF fbHome.Done THEN
            nTestStep := 2;
        END_IF
END_CASE

// --- Test Completion: Assertion & Finish ---
IF nTestStep = 2 THEN
    bCalibrated := fbHome.Done;

    // Assert the axis is marked homed (calibrated)
    AssertEquals_BOOL(
        Expected := TRUE,
        Actual := fbAxisRef[1].Status.Homed,
        Message := 'Axis not calibrated #1'
    );

    // Assert the position matches expected
    AssertEquals_LREAL(
        Delta := 0.001,
        Expected := fExpectedPosition,
        Actual := fbAxisRef[1].NcToPlc.ActPos,
        Message := 'Position is not the expected #2'
    );
    TEST_FINISHED();

ELSIF fbTestTimer.Q THEN
    AssertTrue(
        Condition := FALSE,
        Message := CONCAT('Timed out at step: ', TO_STRING(nTestStep))
    );
    TEST_FINISHED();
END_IF
END_METHOD

METHOD PRIVATE GivenHomeCmdBacklashCompensationInactiveThenMoveStartandCompletesWithBacklashCompensationDisabled_Test2
VAR_INST

    // Subjects under tests
    fbBacklashCompensation : FB_BacklashCompensationNC(
		AxisRef := fbAxisRef[2], 
		iMotionLogger:= fbMotionLogger[2]
	);

    fbHome : FB_HomeNC(
		AxisRef:=fbAxisRef[2],
		iLimSwStatus:=fbLimSwStatus[2],
		iMotionLogger:=fbMotionLogger[2]
	):=(Mode:=E_EpicsHomeCmd.HIGH_LIMIT);

    fbTestTimer : TON := (PT := T#5S, IN := TRUE);
    nTestStep : INT;
    fbCamSwitchPulserSearch: TON := (IN:=TRUE, PT:=T#100MS);
    fbCamSwitchPulserSync: TON := (PT:=T#500MS);
    bHomingOverride: BOOL := TRUE;

END_VAR
TEST(__POUNAME());

// Directional enables must always be TRUE during homing via override.
// 'bHomingOverride' should be TRUE while homing is active.
fbPower[2].Power(
    Enable := TRUE,
    Enable_Positive := bHomingOverride OR fbLimSwStatus[2].LimitForwardEnable,
    Enable_Negative := bHomingOverride OR fbLimSwStatus[2].LimitBackwardEnable,
    Override := 100
);

// == State Machine ==
CASE nTestStep OF
    0: // Enable backlash compensation, but it must be suppressed when homing
        fbBacklashCompensation.EnableBacklashCompensation(UserEnable := TRUE, Compensation := 1.0);
        nTestStep := 1;
    1: // Wait for power enable before issuing home command
        IF fbPower[2].PowerIsEnabled THEN
			fbBacklashCompensation.BacklashCompensation(Enable := FALSE, RampVelo := 10.0);
            // Set override for homing
            bHomingOverride := TRUE;
            // Initiate homing sequence
            fbHome.Home(
				Position := 20.0,
				BufferMode := MC_BufferMode.MC_Aborting,
				HomeMode:=E_EpicsHomeCmd.HIGH_LIMIT
			);
            nTestStep := 2;
        END_IF
    2: // Wait until homing is busy (started)
        IF fbHome.Busy THEN
            AssertFalse(
                Condition := fbBacklashCompensation.Status,
                Message := 'Backlash must be disabled after homing started #2'
            );
            nTestStep := 3;
        END_IF
    3: // Simulate forward cam switch pulse for homing
        IF fbCamSwitchPulserSearch.Q THEN
            fbLimSwStatus[2].LimitForwardEnable := FALSE;
            fbCamSwitchPulserSearch.IN := FALSE;
            fbCamSwitchPulserSync.IN := TRUE;
            nTestStep := 4;
        END_IF
    4: // Simulate cam switch releasing back to TRUE
        IF fbCamSwitchPulserSync.Q THEN
            fbLimSwStatus[2].LimitForwardEnable := TRUE;
            nTestStep := 5;
        END_IF
    5: // When homing is done, stop override
        IF fbHome.Done THEN
            bHomingOverride := FALSE;
            nTestStep := 6;
        END_IF
END_CASE

// -- Cyclic calls to all dependencies --
fbAxisRef[2].ReadStatus();
fbBacklashCompensation();
fbHome();
fbCamSwitchPulserSearch();
fbCamSwitchPulserSync();
fbTestTimer();

// -- Assertion and test finish --
IF nTestStep = 6 THEN
    AssertTrue(
        Condition := (fbAxisRef[2].NcToPlc.ActPos - fbAxisRef[2].NcToPlc.ActPosWithoutPosCorrection) = 0,
        Message := 'Backlash compensation must be enabled #3'
    );
    TEST_FINISHED();

ELSIF fbTestTimer.Q THEN
    AssertTrue(
        Condition := FALSE,
        Message := CONCAT('Timed out at step: ', TO_STRING(nTestStep))
    );
    TEST_FINISHED();
END_IF
END_METHOD

METHOD PRIVATE GivenHomeCmdHomeViaHighModeAndHomeSwPulseThenMoveToUserDefineOffset_Test3
VAR_INST
    fbHome : FB_HomeNC(
		AxisRef:=fbAxisRef[3],
		iLimSwStatus:=fbLimSwStatus[3],
		iMotionLogger:=fbMotionLogger[3]
	) := ( Mode:=E_EpicsHomeCmd.HOME_VIA_HIGH );
	
    fbTestTimer: TON := (IN:=TRUE, PT:=T#5S);
    fbCamSwitchPulserSearch: TON := (IN:=TRUE, PT:=T#500MS);
    fbCamSwitchPulserSync: TON := (PT:=T#1000MS);
    nTestStep : INT;
    fExpectedPosition : LREAL := 20.0;
    fActPosition : LREAL;
    bCalibrated: BOOL;
    // reset this when error or homeDone
    bHomingOverride : BOOL := TRUE;

END_VAR
TEST(__POUNAME());

// Cyclic block calls
fbLimSwStatus[3]();
fbMotionLogger[3]();

fbPower[3].Power(
    Enable := TRUE,
    Enable_Positive := bHomingOverride OR fbLimSwStatus[3].LimitForwardEnable,
    Enable_Negative := bHomingOverride OR fbLimSwStatus[3].LimitBackwardEnable,
    Override := 100.0
);

CASE nTestStep OF
    0:
        IF fbPower[3].PowerIsEnabled THEN
            // Initiate Home command when power is ready
			 fbHome.Home(
					Position := fExpectedPosition,
					BufferMode := MC_BufferMode.MC_Aborting,
					HomeMode:=E_EpicsHomeCmd.HOME_VIA_HIGH
			);
            nTestStep := 1;
        END_IF
    1:
        // Simulate forward cam switch pulse for homing
        IF fbCamSwitchPulserSearch.Q THEN
            fbLimSwStatus[3].LimitHome := TRUE;
            fbCamSwitchPulserSearch.IN := FALSE;
            fbCamSwitchPulserSync.IN := TRUE;
            nTestStep := 2;
        END_IF
    2:
        // Clear home limit after sync pulse
        IF fbCamSwitchPulserSync.Q THEN
            fbLimSwStatus[3].LimitHome := FALSE;
            nTestStep := 3;
        END_IF
    3:
        // Wait for the home sequence to finish
        IF fbHome.Done THEN
            nTestStep := 4;
        END_IF
END_CASE

// Cyclic calls
fbAxisRef[3].ReadStatus();
fbPower[3]();
fbHome();
fbCamSwitchPulserSearch();
fbCamSwitchPulserSync();
fbTestTimer();

IF nTestStep = 4 THEN
    bCalibrated := fbHome.Done;
    AssertEquals_BOOL(
        Expected := TRUE,
        Actual := fbAxisRef[3].Status.Homed,
        Message := 'Axis not calibrated #1'
    );
    AssertEquals_LREAL(
        Delta := 0.001,
        Expected := fExpectedPosition,
        Actual := fbAxisRef[3].NcToPlc.ActPos,
        Message := 'Position is not the expected #2'
    );
    TEST_FINISHED();

ELSIF fbTestTimer.Q THEN
    AssertTrue(
        Condition := FALSE,
        Message := CONCAT('Timed out at step: ', TO_STRING(nTestStep))
    );
    TEST_FINISHED();
END_IF
END_METHOD

METHOD PRIVATE GivenHomeCmdHomeViaHighModeForwardSwPulseBeforeHomeSwPulseThenMoveToUserDefineOffset_Test4
VAR_INST
    fbHome : FB_HomeNC(
		AxisRef:=fbAxisRef[4],
		iLimSwStatus:=fbLimSwStatus[4],
		iMotionLogger:=fbMotionLogger[4]
	) := ( Mode := E_EpicsHomeCmd.HOME_VIA_HIGH );
	
    fbTestTimer: TON := (IN:=TRUE, PT:=T#5S);
    fbCamSwitchPulserSearch: TON := (IN:=TRUE, PT:=T#500MS);
    fbCamSwitchPulserSync: TON := (PT:=T#1000MS);
    nTestStep : INT;
    fExpectedPosition : LREAL := 20.0;
    fActPosition : LREAL;
    bCalibrated: BOOL;
    // reset this when error or homeDone
    bHomingOverride : BOOL := TRUE;
END_VAR
TEST(__POUNAME());

// Cyclic preparation and block invocation
fbAxisRef[4].ReadStatus();
fbLimSwStatus[4]();
fbMotionLogger[4]();
fbPower[4].Power(
    Enable := TRUE,
    Enable_Positive := bHomingOverride OR fbLimSwStatus[4].LimitForwardEnable,
    Enable_Negative := bHomingOverride OR fbLimSwStatus[4].LimitForwardEnable, // Note: both positive and negative use ForwardEnable here
    Override := 100.0
);

